			// Zyklisch auf neue Daten pollen
			fbReceiveDataBytes(
				pPrefix				:= ADR(stOptionsIntern.sPrefix),
				LenPrefix			:= stOptionsIntern.nLenPrefix,
				pSuffix				:= ADR(stOptionsIntern.sSuffix),
				LenSuffix			:= stOptionsIntern.nLenSuffix,
				
				Timeout				:= stOptionsIntern.tTimeTimeout,
				Reset					:= FALSE ,
				
				pReceiveData		:= ADR(stRxStringBuffer),
				SizeReceiveData	:= SIZEOF(stRxStringBuffer)-1,
				RXbuffer				:= stRxBuffer
			);

			IF fbReceiveDataBytes.Error <> 0
			THEN	// Fehler beim Datenempfangen
				nRxCount					:= 0;
				bNeueDatenEmpfangen	:= TRUE;
				ccl_Receive.bBusy		:= FALSE;
				ccl_Receive.bDone		:= TRUE;
				ccl_Receive.bError	:= TRUE;
				ccl_Receive.nErrorId	:= fbReceiveDataBytes.Error;
			ELSE

				IF fbReceiveDataBytes.DataReceived
				THEN	// Alle Daten wurden erfolgreich empfangen
				
					nRxCount	:= UDINT_TO_INT(fbReceiveDataBytes.LenReceiveData);
					IF nRxCount <= cBufferSize_StringBuffer
					THEN
						stRxStringBuffer.sData:=LEFT(stRxStringBuffer.sData,nRxCount);
					ELSE
						stRxStringBuffer.sData:=LEFT(stRxStringBuffer.sData,cBufferSize_StringBuffer);
					END_IF
					stRxStringBuffer:= nccl_ReceiveBarcode(stRxStringBuffer);
					nRxCount:=LEN(stRxStringBuffer.sData);

					bRxTimeout:= fbReceiveDataBytes.RxTimeout;
					bNeueDatenEmpfangen	:= TRUE;
				END_IF;
			END_IF
	END_CASE

	// Empfang Oberflaeche. Darauf warten, die die Oberfäche das Bit zurück setzt.
	IF	bNeueDatenEmpfangen
		AND stOptions.nCommVB = 1
	THEN
		bWartenAufVBA_HMI	:= TRUE;
	END_IF

END_IF
END_METHOD

METHOD FB_init : BOOL
VAR_INPUT
	bInitRetains	: BOOL; // if TRUE, the retain variables are initialized (warm start / cold start)
	bInCopyCode		: BOOL;  // if TRUE, the instance afterwards gets moved into the copy code (online change)
	
	I_Options		: ST_ComPortOptions;	
END_VAR
stOptions	:= I_Options;
END_METHOD

METHOD PUBLIC nccl_Config : ST_MethodResult	// Methode muss so lange aufgerufen werden, bis True zurück gibt
// Konfigruation der Klemmen

CASE stOptions.ePort OF
	// PC-ComPort kann man nicht aus der PLC heraus konfigurieren
	E_ComPortHardware.cComportPc:
	
		nccl_Config.bDone	:= TRUE;

	// EL-Klemmen Konfigurieren
	E_ComPortHardware.cComportEL:
	
		CASE nConfigState OF
			
			0:  // Baudrate schreiben, dafür wird mit nWordBuffer die Zeile der Dropdownliste errechnet, die dann geschrieben wird. Es wird nicht direkt die Baudrate geschrieben.(Wäre ja auch zu einfach)
				nccl_Config.bBusy	:= TRUE;
				nIndex:=16#4073;
				nSubIndex:=0;

				nWordBuffer	:= 4;
				nTmpVar		:= stOptions.nBaudrate;
				
				// Ist die Baudrate bei min(1200) angelangt, ist fertig berechnet
				WHILE nTmpVar > 2400 DO
					nTmpVar		:= nTmpVar/2;
					nWordBuffer	:= nWordBuffer+1;
				END_WHILE

				fbEcCoWrite(
					sNetId		:= F_CreateAmsNetId(stComPortIn.stInfoData.stADSNetId) ,
					nSlaveAddr	:= stComPortIn.stInfoData.nADSPort,

					nSubIndex	:= nSubIndex,
					nIndex		:= nIndex,

					pSrcBuf		:= ADR(nWordBuffer),
					cbBufLen		:= SIZEOF(nWordBuffer),
					bExecute		:= NOT fbEcCoWrite.bBusy,
					tTimeout		:= T#3S
				);

			1:  // Frame
				nccl_Config.bBusy	:= TRUE;
				nIndex:=16#4074;
				nSubIndex:=0;

				IF stOptions.nDatenbits = 7
				THEN
					IF stOptions.nStopbits = 1
					THEN
						(*7x1 *)
						CASE stOptions.nParitaet OF
							PARITY_NONE	: nWordBuffer	:= 1;
							PARITY_EVEN	: nWordBuffer	:= 1;
							PARITY_ODD	: nWordBuffer	:= 2;
						END_CASE
					ELSE
						(*7x2 *)
						CASE stOptions.nParitaet OF
							PARITY_NONE	: nWordBuffer	:= 9;
							PARITY_EVEN	: nWordBuffer	:= 9;
							PARITY_ODD	: nWordBuffer	:= 10;
						END_CASE
					END_IF
				ELSE
					(*8x1 *)
					IF stOptions.nStopbits = 1 THEN
						CASE stOptions.nParitaet OF
							PARITY_NONE	: nWordBuffer	:= 3;
							PARITY_EVEN	: nWordBuffer	:= 4;
							PARITY_ODD	: nWordBuffer	:= 5;
						END_CASE
					ELSE
						(*8x2 *)
						CASE stOptions.nParitaet OF
							PARITY_NONE	: nWordBuffer	:= 11;
							PARITY_EVEN	: nWordBuffer	:= 12;
							PARITY_ODD	: nWordBuffer	:= 13;
						END_CASE
					END_IF
				END_IF

				fbEcCoWrite(
					sNetId		:= F_CreateAmsNetId(stComPortIn.stInfoData.stADSNetId) ,
					nSlaveAddr	:= stComPortIn.stInfoData.nADSPort,

					nSubIndex	:= nSubIndex,
					nIndex		:= nIndex,

					pSrcBuf		:= ADR(nWordBuffer),
					cbBufLen		:= SIZEOF(nWordBuffer),
					bExecute		:= NOT fbEcCoWrite.bBusy,
					tTimeout		:= T#3S
				);

			2:  // Handshake RTS/CTS
				nccl_Config.bBusy	:= TRUE;
				nIndex		:= 16#4075;
				nSubIndex	:= 1;

				IF stOptions.nHandshake = HANDSHAKE_RTSCTS
				THEN
					bBuffer:=TRUE;
				ELSE
					bBuffer:=FALSE;
				END_IF

				fbEcCoWrite(
					sNetId		:= F_CreateAmsNetId(stComPortIn.stInfoData.stADSNetId) ,
					nSlaveAddr	:= stComPortIn.stInfoData.nADSPort,

					nSubIndex	:= nSubIndex,
					nIndex		:= nIndex,

					pSrcBuf		:= ADR(bBuffer),
					cbBufLen		:= SIZEOF(bBuffer),
					bExecute		:= NOT fbEcCoWrite.bBusy,
					tTimeout		:= T#3S
				);

			3:  (* XON/XOFF tx *)
				nccl_Config.bBusy	:= TRUE;
				nIndex		:= 16#4075;
				nSubIndex	:= 2;

				IF stOptions.nHandshake = HANDSHAKE_XONXOFF
				THEN
					bBuffer:=TRUE;
				ELSE
					bBuffer:=FALSE;
				END_IF

				fbEcCoWrite(
					sNetId		:= F_CreateAmsNetId(stComPortIn.stInfoData.stADSNetId) ,
					nSlaveAddr	:= stComPortIn.stInfoData.nADSPort,

					nSubIndex	:= nSubIndex,
					nIndex		:= nIndex,

					pSrcBuf		:= ADR(bBuffer),
					cbBufLen		:= SIZEOF(bBuffer),
					bExecute		:= NOT fbEcCoWrite.bBusy,
					tTimeout		:= T#3S
				);

			4:  (* XON/XOFF rx *)
				nccl_Config.bBusy	:= TRUE;
				nIndex		:= 16#4075;
				nSubIndex	:= 3;

				IF stOptions.nHandshake = HANDSHAKE_XONXOFF
				THEN
					bBuffer	:= TRUE;
				ELSE
					bBuffer	:= FALSE;
				END_IF

				fbEcCoWrite(
					sNetId		:= F_CreateAmsNetId(stComPortIn.stInfoData.stADSNetId) ,
					nSlaveAddr	:= stComPortIn.stInfoData.nADSPort,

					nSubIndex	:= nSubIndex,
					nIndex		:= nIndex,

					pSrcBuf		:= ADR(bBuffer),
					cbBufLen		:= SIZEOF(bBuffer),
					bExecute		:= NOT fbEcCoWrite.bBusy,
					tTimeout		:= T#3S
				);
				
		END_CASE

		IF NOT fbEcCoWrite.bBusy
		THEN
			// Bei Fehler ErrorId speichern und Config abbrechen
			IF fbEcCoWrite.bError
			THEN
				nccl_Config.nErrorId	:= UDINT_TO_INT(fbEcCoWrite.nErrId);
			ELSE
				IF nConfigState < 4
				THEN
					nConfigState	:= nConfigState+1;
				ELSE
					nccl_Config.bBusy	:= FALSE;
					nccl_Config.bDone	:= TRUE;	// Konfiguration ist fertig!!!
				END_IF
			END_IF

		END_IF
		
		nccl_Config.bError	:= fbEcCoWrite.bError;
		nccl_Config.nErrorId	:= UDINT_TO_INT(fbEcCoWrite.nErrId);

	// KL-Klemmen Konfigurieren
	E_ComPortHardware.cComportKL:
	
		CASE stOptions.eComPortBytes OF
			
			E_ComPortKlemmenBytes.cComport3Bytes:
			
				fbComPortKL6configuration(
					Execute		:= NOT fbComPortKL6configuration.Busy,
					Mode			:= SERIALLINEMODE_KL6_3B_ALTERNATIVE,
					Baudrate		:= stOptions.nBaudrate,
					NoDatabits	:= UDINT_TO_BYTE(stOptions.nDatenbits),
					Parity		:= stOptions.nParitaet,
					Stopbits		:= UDINT_TO_BYTE(stOptions.nStopbits),
					Handshake	:= stOptions.nHandshake,
					pCOMin		:= ADR(stComPortIn.stKlemmeIn3B),
					pCOMout		:= ADR(stComPortOut.stKlemmeOut3B),
					SizeComIn	:= SIZEOF(stComPortIn.stKlemmeIn3B)
				);
				
				nccl_Config.bBusy		:= fbComPortKL6configuration.Busy;
				nccl_Config.bDone		:= fbComPortKL6configuration.Done;
				nccl_Config.bError	:= fbComPortKL6configuration.Error;
				nccl_Config.nErrorId	:= fbComPortKL6configuration.ErrorId;

			E_ComPortKlemmenBytes.cComport5Bytes:
			
				fbComPortKL6configuration(
					Execute		:= NOT fbComPortKL6configuration.Busy ,
					Mode			:= SERIALLINEMODE_KL6_5B_STANDARD,
					Baudrate		:= UINT_TO_UDINT(stOptions.nBaudrate),
					NoDatabits	:= UDINT_TO_BYTE(stOptions.nDatenbits),
					Parity		:= stOptions.nParitaet,
					Stopbits		:= UDINT_TO_BYTE(stOptions.nStopbits),
					Handshake	:= stOptions.nHandshake,
					pCOMin		:= ADR(stComPortIn.stKlemmeIn5B),
					pCOMout		:= ADR(stComPortOut.stKlemmeOut5B),
					SizeComIn	:= SIZEOF(stComPortIn.stKlemmeIn5B)
				);
				
				nccl_Config.bBusy		:= fbComPortKL6configuration.Busy;
				nccl_Config.bDone		:= fbComPortKL6configuration.Done;
				nccl_Config.bError	:= fbComPortKL6configuration.Error;
				nccl_Config.nErrorId	:= fbComPortKL6configuration.ErrorId;

			E_ComPortKlemmenBytes.cComport22Bytes:
			
				fbComPortKL6configuration(
					Execute		:= NOT fbComPortKL6configuration.Busy ,
					Mode 			:= SERIALLINEMODE_KL6_22B_STANDARD,
					Baudrate		:= UDINT_TO_UINT(stOptions.nBaudrate),
					NoDatabits	:= UDINT_TO_BYTE(stOptions.nDatenbits),
					Parity		:= stOptions.nParitaet,
					Stopbits		:= UDINT_TO_BYTE(stOptions.nStopbits),
					Handshake	:= stOptions.nHandshake,
					pCOMin		:= ADR(stComPortIn.stKlemmeIn22B),
					pCOMout		:= ADR(stComPortOut.stKlemmeOut22B),
					SizeComIn	:= SIZEOF(stComPortIn.stKlemmeIn22B)
				);
				
				nccl_Config.bBusy		:= fbComPortKL6configuration.Busy;
				nccl_Config.bDone		:= fbComPortKL6configuration.Done;
				nccl_Config.bError	:= fbComPortKL6configuration.Error;
				nccl_Config.nErrorId	:= fbComPortKL6configuration.ErrorId;

		END_CASE
END_CASE;

// Konfiguration in die internen Konfiguration übernehmen
stOptionsIntern.tTimeTimeout	:= UDINT_TO_TIME(stOptions.nTimeout);

// Präfix-Konfiguration
stOptionsIntern.nLenPrefix	:= 0;
stOptionsIntern.sPrefix		:= '';

stOptionsIntern.nPrefix		:= UDINT_TO_BYTE(stOptions.nPrefix);

IF stOptionsIntern.nPrefix > 0
THEN
	stOptionsIntern.nLenPrefix	:= stOptionsIntern.nLenPrefix+1;
	stOptionsIntern.sPrefix		:= CONCAT(stOptionsIntern.sPrefix,CHR(stOptionsIntern.nPrefix));
END_IF

// Suffix-Konfiguration
stOptionsIntern.nLenSuffix	:= 0;
stOptionsIntern.sSuffix		:= '';

stOptionsIntern.arrSuffix[1]	:= UDINT_TO_BYTE(stOptions.nSuffix1);
IF stOptionsIntern.arrSuffix[1] > 0
THEN
	stOptionsIntern.nLenSuffix	:= stOptionsIntern.nLenSuffix+1;
	stOptionsIntern.sSuffix		:= CONCAT(stOptionsIntern.sSuffix,CHR(stOptionsIntern.arrSuffix[1]));
END_IF

stOptionsIntern.arrSuffix[2]	:= UDINT_TO_BYTE(stOptions.nSuffix2);
IF stOptionsIntern.arrSuffix[2] > 0
THEN
	stOptionsIntern.nLenSuffix	:= stOptionsIntern.nLenSuffix+1;
	stOptionsIntern.sSuffix		:= CONCAT(stOptionsIntern.sSuffix,CHR(stOptionsIntern.arrSuffix[2]));

	IF stOptionsIntern.arrSuffix[1] = 0
	THEN
		stOptionsIntern.arrSuffix[1]:= stOptionsIntern.arrSuffix[2];
		stOptionsIntern.arrSuffix[2]:= 0;
	END_IF
END_IF

// Bufferlänge auf bei Überschreiten der max Größe, auf die max Größe setzen
IF stOptions.nLength > cBufferSize_IntBuffer
	OR stOptions.nLength = 0
THEN
	stOptionsIntern.nLength:=cBufferSize_IntBuffer;
ELSE
	stOptionsIntern.nLength:=stOptions.nLength;
END_IF
END_METHOD

METHOD INTERNAL nccl_PrepareSendBarcode : ST_ComPortStringBuffer
VAR_INPUT
	I_stSendString	:	ST_ComPortStringBuffer;
END_VAR
IF stOptionsIntern.nLenPrefix > 0
THEN
	nccl_PrepareSendBarcode.sData:=CONCAT(stOptionsIntern.sPrefix,I_stSendString.sData);
ELSE
	nccl_PrepareSendBarcode	:= I_stSendString;
END_IF

IF stOptionsIntern.nLenSuffix > 0
THEN
	nccl_PrepareSendBarcode.sData:=CONCAT(nccl_PrepareSendBarcode.sData,stOptionsIntern.sSuffix);
END_IF
END_METHOD

METHOD INTERNAL nccl_ReceiveBarcode : ST_ComPortStringBuffer
VAR_INPUT
	I_stReceiveString	: ST_ComPortStringBuffer;
END_VAR

VAR
	nStartPosition	: INT;
	nEndPosition	: INT;
	bPrefixFound	: BOOL;
END_VAR
nStartPosition	:= 0;
IF stOptionsIntern.nLenPrefix = 0
THEN
	bPrefixFound:=TRUE;
ELSE
	bPrefixFound:=FALSE;

	REPEAT
		nStartPosition	:= FIND(I_stReceiveString.sData,stOptionsIntern.sPrefix);
		IF nStartPosition > 0
		THEN
			bPrefixFound:=TRUE; (* Mindesten 1 x Prefix *)

			nStartPosition	:= nStartPosition + stOptionsIntern.nLenPrefix;
			I_stReceiveString.sData	:= MID(I_stReceiveString.sData,LEN(I_stReceiveString.sData)-nStartPosition+1,nStartPosition);
		END_IF
	UNTIL
		nStartPosition = 0
	END_REPEAT
END_IF

IF bPrefixFound
THEN
	nEndPosition:=0;

	IF stOptionsIntern.nLenSuffix = 0
	THEN
		nEndPosition	:= LEN(I_stReceiveString.sData);
	ELSE
		nEndPosition	:= FIND(I_stReceiveString.sData,stOptionsIntern.sSuffix)-1;
	END_IF

	IF nEndPosition > 0
	THEN
		nccl_ReceiveBarcode.sData	:= MID(I_stReceiveString.sData,nEndPosition,1);
	END_IF
END_IF
END_METHOD

METHOD PUBLIC nccl_Reset : BOOL
VAR
	nRxBufferIndx	: INT;
	fbClearBuffer	: ClearComBuffer;
END_VAR
// Reset
IF NOT stConfigResult.bBusy
THEN
	bNeueDatenEmpfangen	:= FALSE;
	bWartenAufVBA_HMI		:= FALSE;
	bRxTimeout				:=FALSE;

	// Empfangsdaten löschen
	FOR nRxBufferIndx	:= 0 TO cBufferSize_IntBuffer
	DO
		stRxIntBuffer.arrData[nRxBufferIndx]:=0;
	END_FOR

	stRxStringBuffer.sData:='';
	
	// internen Empfangspuffer löschen
	fbClearBuffer(Buffer:=stRxBuffer);

	// Empfangsbaustein für Datenstream resetten
	fbReceiveDataBytes(
		Reset				:= TRUE ,
		pReceiveData	:= ADR(stRxByteBuffer),
		RXbuffer			:= stRxBuffer
	);

	// interne Empfangs- und Sendepuffer nochmals händisch löschen- 
	stTxBuffer.Count:=0;
	stTxBuffer.RdIdx:=0;
	stTxBuffer.WrIdx:=0;
	stTxBuffer.Error:=0;

	stRxBuffer.Count:=0;
	stRxBuffer.RdIdx:=0;
	stRxBuffer.WrIdx:=0;
	stRxBuffer.Error:=0;

	// Diagnose zurücksetzen
	nDiagRxCycleCounter	:=0;
	nDiagRxErrorCounter	:=0;
	nDiagRxLastErrorId	:=0;
	nDiagRxDataCounter	:=0;

	sTmpDiagMessage	:= CONCAT('RxCycle:', UINT_TO_STRING(nDiagRxCycleCounter));
	sTmpDiagMessage	:= CONCAT(sTmpDiagMessage, CONCAT(' - RxData:', INT_TO_STRING(nDiagRxDataCounter)));
	sTmpDiagMessage	:= CONCAT(sTmpDiagMessage, CONCAT(' - RxError:', UINT_TO_STRING(nDiagRxErrorCounter)));
	sTmpDiagMessage	:= CONCAT(sTmpDiagMessage, CONCAT(' - RxErrorId:', INT_TO_STRING(nDiagRxLastErrorId)));
	sDiagMessage		:= sTmpDiagMessage;

	bStartPLC	:= FALSE;	// Config auslösen
	nccl_Reset	:= TRUE;	// Resetten fertig
END_IF
END_METHOD

{attribute 'hide_all_locals'}
METHOD PUBLIC nccl_Send : ST_MethodResult	// Methode ist innerhalb eines Zyklusses fertig.
VAR_INPUT
	I_stTxIntBuffer			: ST_ComPortIntBuffer;	// Int Uebergabepuffer
	I_stTxStringBuffer		: ST_ComPortStringBuffer;	// String Uebergabepuffer

	I_nTxCount					: INT;	// Anzahl zu sendender Zeichen
	I_eTxProtokoll				: E_ComPortProtokoll	:= E_ComPortProtokoll.cProtokollNone;	// Sendenprotokoll
END_VAR
VAR
	nTxBufferIndx				: INT;
	stBarcodeTxStringBuffer	: ST_ComPortStringBuffer;
	
	eProtokoll					: E_ComPortProtokoll;
	stTxByteBuffer				: Tc2_SerialCom.P3964buffer;
	fbSendByteDirect			: Tc2_SerialCom.SendByte;
	fbSendDataBytes			: Tc2_SerialCom.SendData;
END_VAR
// Senden
IF stOptions.nAktiv = 1
	AND NOT stConfigResult.bBusy
THEN
	nccl_Send.bBusy	:= TRUE;	// pauschal auf busy setzen

	IF I_eTxProtokoll <> E_ComPortProtokoll.cProtokollNone
	THEN
		eProtokoll := I_eTxProtokoll;
	ELSE
		eProtokoll := stOptions.eProtokoll;
	END_IF

	CASE eProtokoll OF
		E_ComPortProtokoll.cProtokollNone:
			;	// Ohne Protokoll nix machen
			
		E_ComPortProtokoll.cProtokollData:
			
			nTxBufferIndx:=0;
			WHILE nTxBufferIndx < I_nTxCount
				AND nTxBufferIndx <= cBufferSize_IntBuffer
			DO
				stTxByteBuffer.D[nTxBufferIndx]	:= UINT_TO_BYTE(I_stTxIntBuffer.arrData[nTxBufferIndx]);
				nTxBufferIndx	:= nTxBufferIndx+1;
			END_WHILE

			fbSendDataBytes(
				pSendData:= ADR(stTxByteBuffer),
				Length	:= INT_TO_UDINT(I_nTxCount),
				TXbuffer	:= stTxBuffer);

			// Sendefehler
			IF  fbSendDataBytes.Error <> 0
			THEN
				nccl_Send.nErrorId	:= fbSendDataBytes.Error;
				nccl_Send.bError	:= TRUE; 
				nccl_Send.bBusy	:= FALSE;
			ELSE	// Erfolgreich gesendet
				IF NOT fbSendDataBytes.Busy
				THEN
					nccl_Send.bBusy	:= FALSE;
					nccl_Send.bDone	:= TRUE;
				END_IF
			END_IF

		E_ComPortProtokoll.cProtokollDirect:
			
			nTxBufferIndx := 0;
			IF I_nTxCount > cBufferSize_IntBuffer
			THEN
				I_nTxCount := cBufferSize_IntBuffer;
			END_IF

			WHILE nTxBufferIndx < I_nTxCount
				AND fbSendByteDirect.Error = 0
			DO
				fbSendByteDirect(
					SendByte	:= UINT_TO_BYTE(I_stTxIntBuffer.arrData[nTxBufferIndx]),
					TXbuffer	:= stTxBuffer
				);
				nTxBufferIndx	:= nTxBufferIndx+1;
				
			END_WHILE

			// Sendefehler
			IF  fbSendByteDirect.Error <> 0
			THEN
				nccl_Send.nErrorId	:= fbSendByteDirect.Error;
				nccl_Send.bError	:= TRUE; 
				nccl_Send.bBusy	:= FALSE;
			ELSE	// Erfolgreich gesendet
				IF NOT fbSendByteDirect.Busy
				THEN
					nccl_Send.bBusy	:= FALSE;
					nccl_Send.bDone	:= TRUE;
				END_IF
			END_IF

		E_ComPortProtokoll.cProtokollBarcode:
			
			stBarcodeTxStringBuffer	:= nccl_PrepareSendBarcode(I_stTxStringBuffer);

			fbSendDataBytes(
				pSendData	:= ADR(stBarcodeTxStringBuffer),
				Length		:= INT_TO_BYTE(LEN(stBarcodeTxStringBuffer.sData)),
				TXbuffer		:= stTxBuffer);

			// Sendefehler
			IF  fbSendDataBytes.Error <> 0
			THEN
				nccl_Send.nErrorId	:= fbSendDataBytes.Error;
				nccl_Send.bError		:= TRUE; 
				nccl_Send.bBusy		:= FALSE;
			ELSE	// Erfolgreich gesendet
				IF NOT fbSendDataBytes.Busy
				THEN
					nccl_Send.bBusy	:= FALSE;
					nccl_Send.bDone	:= TRUE;
				END_IF
			END_IF
	END_CASE
END_IF

stSendResult	:= nccl_Send;
END_METHOD

PROPERTY PUBLIC P_bDatenVorhanden : BOOL
GET
P_bDatenVorhanden	:= bNeueDatenEmpfangen;
END_GET
END_PROPERTY

// Liest die Empfangenen Daten aus und setzt das Empfangsbit zurück
PROPERTY PUBLIC P_stEmpfangeneDaten : ST_ComPortIntBuffer
GET
P_stEmpfangeneDaten	:= stRxIntBuffer;
bNeueDatenEmpfangen	:= FALSE;
END_GET
END_PROPERTY

// Liest die Empfangenen Daten aus und setzt das Empfangsbit zurück
PROPERTY PUBLIC P_stEmpfangenerString : STRING
GET
P_stEmpfangenerString	:= stRxStringBuffer.sData;
bNeueDatenEmpfangen		:= FALSE;
END_GET
END_PROPERTY

END_FUNCTION_BLOCK

// POUs/DiagSafety/FB_DiagEL2904
// OBSOLET, wenn man FB_TwinSAFEKlemmenInfo benutzt
FUNCTION_BLOCK FB_DiagEL2904
VAR_INPUT
	I_stEcAdsAddr			: AMSADDR;
	I_nDiag					: USINT;
	I_strBMK					: STRING;
END_VAR
VAR_OUTPUT
	Q_stTemperatur 		: ST_EL2904Temp;
	Q_bError					: BOOL;
	Q_strDiag				: STRING;
END_VAR
VAR
	nStep					: INT;
	nLastStep			: INT;
	tonReadDiag			: TON;
	fbEcCoeSdoRead		: FB_EcCoESdoReadEx;
	stDiagObject		: ST_EL2904Diag;
	nDiag0_3				: BYTE;
	strDiag				: STRING;
END_VAR


act_Diag();
act_DiagObjekte();

IF strDiag <> ''
THEN
	Q_strDiag 	:= CONCAT(I_strBMK,CONCAT(' ',strDiag));
	Q_bError		:= TRUE;
ELSE
	Q_bError		:= FALSE;
END_IF

ACTION act_Diag:

strDiag:='';

IF I_nDiag.4 
THEN
	strDiag	:= 'Fehler beim FSoE Slave erkannt | '; 
END_IF

IF I_nDiag.5 
THEN
	strDiag	:= CONCAT(strDiag,'FSoE Slave meldet Failsafe Value aktiv | ');
END_IF

IF I_nDiag.6 
THEN
	strDiag	:= CONCAT(strDiag,'StartUp | ');
END_IF

IF I_nDiag.7 
THEN
	strDiag	:= CONCAT(strDiag, 'FSoE Master meldet Failsafe Value aktiv | ');
END_IF
	
nDiag0_3 := USINT_TO_BYTE(I_nDiag) AND 16#0F;

CASE nDiag0_3 OF
	1:		strDiag	:= CONCAT(strDiag,'Ungültiges Kommando | ');
	2:		strDiag	:= CONCAT(strDiag,'Unbekanntes Kommando | ');
	3:		strDiag	:= CONCAT(strDiag,'Ungültige Connection ID | ');
	4:		strDiag	:= CONCAT(strDiag,'Ungültige CRC | ');
	5:		strDiag	:= CONCAT(strDiag,'Watchdog abgelaufen | ');
	6:		strDiag	:= CONCAT(strDiag,'Ungültige FSoE Adresse | ');
	7:		strDiag	:= CONCAT(strDiag,'Ungültige Daten | ');
	8:		strDiag	:= CONCAT(strDiag,'Ungültige Kommunikationsparameterlänge | ');
	9:		strDiag	:= CONCAT(strDiag,'Ungültige Kommunikationsparameter | ');
	10:	strDiag	:= CONCAT(strDiag,'Ungültige Anwenderparameterlänge | ');
	11:	strDiag	:= CONCAT(strDiag,'Ungültige Anwenderparameter | ');
	12:	strDiag	:= CONCAT(strDiag,'FSoE Master Reset | ');
	13:	strDiag	:= CONCAT(strDiag,'Modulfehler auf Slave erkannt, bei aktivierter Option "Modulfehler ist ComError" | ');
	14:	strDiag	:= CONCAT(strDiag,'Modulfehler auf EL290x erkannt, bei aktivierter Option "Error acknowledge active" | ');
	15:	strDiag	:= CONCAT(strDiag,'Slave noch nicht gestartet, oder unerwartetes Fehlerargument | ');
END_CASE

IF stDiagObject.nErrorOutputs.0
THEN
	strDiag	:= CONCAT(strDiag,'Fremdeinspeisung oder Querschluss am Ausgang 1');
ELSIF  stDiagObject.nErrorOutputs.1 
THEN
	strDiag	:= CONCAT(strDiag,'Fremdeinspeisung oder Querschluss am Ausgang 2');
ELSIF  stDiagObject.nErrorOutputs.2
THEN
	strDiag	:= CONCAT(strDiag,'Fremdeinspeisung oder Querschluss am Ausgang 3');
ELSIF  stDiagObject.nErrorOutputs.3 
THEN
	strDiag	:= CONCAT(strDiag,'Fremdeinspeisung oder Querschluss am Ausgang 4');
ELSIF  stDiagObject.nErrorOutputs.4 
THEN
	strDiag	:= CONCAT(strDiag,'Ausgangsstrom < 20mA oder > 500mA am Ausgang 1');
ELSIF  stDiagObject.nErrorOutputs.5
THEN
	strDiag	:= CONCAT(strDiag,'Ausgangsstrom < 20mA oder > 500mA am Ausgang 2');
ELSIF  stDiagObject.nErrorOutputs.6 
THEN
	strDiag	:= CONCAT(strDiag,'Ausgangsstrom < 20mA oder > 500mA am Ausgang 3');
ELSIF  stDiagObject.nErrorOutputs.7 
THEN
	strDiag	:= CONCAT(strDiag,'Ausgangsstrom < 20mA oder > 500mA am Ausgang 4');
	
ELSIF stDiagObject.nSupplyError.0
THEN
	strDiag	:= CONCAT(strDiag,'Feldspannung zu hoch');
ELSIF stDiagObject.nSupplyError.1
THEN
	strDiag	:= CONCAT(strDiag,'Feldspannung zu niedrig');
	
ELSIF stDiagObject.nTemperatureError.0
THEN
	strDiag	:= CONCAT(strDiag,'Übertemperatur µC1');
ELSIF stDiagObject.nTemperatureError.1
THEN
	strDiag	:= CONCAT(strDiag,'Übertemperatur µC2');
ELSIF stDiagObject.nTemperatureError.2
THEN
	strDiag	:= CONCAT(strDiag,'Übertemperatur der Ausgangsplatine');
ELSIF stDiagObject.nTemperatureError.3
THEN
	strDiag	:= CONCAT(strDiag,'Untertemperatur µC1');
ELSIF stDiagObject.nTemperatureError.4
THEN
	strDiag	:= CONCAT(strDiag,'Untertemperatur µC2');
ELSIF stDiagObject.nTemperatureError.5
THEN
	strDiag	:= CONCAT(strDiag,'Untertemperatur der Ausgangsplatine');
ELSIF stDiagObject.nTemperatureError.6
THEN
	strDiag	:= CONCAT(strDiag,'Temperaturdifferenz auf der Prozessorplatine zu groß');
ELSIF stDiagObject.nTemperatureError.7
THEN
	strDiag	:= CONCAT(strDiag,'Temperaturdifferenz zwischen den Platinen zu groß');
END_IF
END_ACTION

ACTION act_DiagObjekte:
CASE nStep OF

0: tonReadDiag(IN:= TRUE,	
					PT :=T#2S);
		fbEcCoeSdoRead(
		bExecute			:= FALSE);
	IF tonReadDiag.Q
	THEN
		nStep := 10;
	END_IF

10:	
	fbEcCoeSdoRead(
		sNetId			:= F_CreateAmsNetId(I_stEcAdsAddr.netId), 
		nSlaveAddr		:= I_stEcAdsAddr.port, 
		nSubIndex		:= 1, 
		nIndex			:= 16#FA80, 
		pDstBuf			:= ADR(Q_stTemperatur), 
		cbBufLen			:= SIZEOF(Q_stTemperatur), 
		bExecute			:= TRUE, 
		tTimeout			:= T#5S, 
		bCompleteAccess:= TRUE );
	
	IF NOT fbEcCoeSdoRead.bBusy
		AND NOT fbEcCoeSdoRead.bError
	THEN
		fbEcCoeSdoRead(bExecute := FALSE);
		nStep := 20;
	ELSIF fbEcCoeSdoRead.bError
	THEN
		nStep := 0;
	END_IF

20: fbEcCoeSdoRead(
		sNetId			:= F_CreateAmsNetId(I_stEcAdsAddr.netId), 
		nSlaveAddr		:= I_stEcAdsAddr.port, 
		nSubIndex		:= 1, 
		nIndex			:= 16#800E, 
		pDstBuf			:= ADR(stDiagObject), 
		cbBufLen			:= SIZEOF(stDiagObject), 
		bExecute			:= TRUE, 
		tTimeout			:= T#5S, 
		bCompleteAccess:= TRUE);
	IF NOT fbEcCoeSdoRead.bBusy
		AND NOT fbEcCoeSdoRead.bError
	THEN
		nStep	:= 0;
	ELSIF fbEcCoeSdoRead.bError
	THEN
		nStep := 0;
	END_IF
END_CASE


IF nStep <> nLastStep
THEN
	tonReadDiag(IN:= FALSE);
	nLastStep := nStep;
END_IF
END_ACTION

END_FUNCTION_BLOCK

// POUs/DiagSafety/FB_DiagEL2912
// OBSOLET, wenn man FB_TwinSAFEKlemmenInfo benutzt
FUNCTION_BLOCK FB_DiagEL2912
VAR_INPUT				
	I_stEcAdsAddr			: AMSADDR;
	I_nDiag					: USINT;
	I_strBMK					: STRING;
END_VAR
VAR_OUTPUT
	Q_bError					: BOOL;
	Q_strDiag				: STRING;
END_VAR
VAR
	nDiag0_3				: BYTE;
	strDiag				: STRING;
END_VAR


act_Diag();

IF strDiag <> ''
THEN
	Q_strDiag 	:= CONCAT(I_strBMK,CONCAT(' ',strDiag));
	Q_bError		:= TRUE;
ELSE
	Q_bError		:= FALSE;
END_IF

ACTION act_Diag:

strDiag:='';

IF I_nDiag.4 
THEN
	strDiag	:= 'Fehler beim FSoE Slave erkannt | '; 
END_IF

IF I_nDiag.5 
THEN
	strDiag	:= CONCAT(strDiag,'FSoE Slave meldet Failsafe Value aktiv | ');
END_IF

IF I_nDiag.6 
THEN
	strDiag	:= CONCAT(strDiag,'StartUp | ');
END_IF

IF I_nDiag.7 
THEN
	strDiag	:= CONCAT(strDiag, 'FSoE Master meldet Failsafe Value aktiv | ');
END_IF
	
nDiag0_3 := USINT_TO_BYTE(I_nDiag) AND 16#0F;

CASE nDiag0_3 OF
	1:		strDiag	:= CONCAT(strDiag,'Ungültiges Kommando | ');
	2:		strDiag	:= CONCAT(strDiag,'Unbekanntes Kommando | ');
	3:		strDiag	:= CONCAT(strDiag,'Ungültige Connection ID | ');
	4:		strDiag	:= CONCAT(strDiag,'Ungültige CRC | ');
	5:		strDiag	:= CONCAT(strDiag,'Watchdog abgelaufen | ');
	6:		strDiag	:= CONCAT(strDiag,'Ungültige FSoE Adresse | ');
	7:		strDiag	:= CONCAT(strDiag,'Ungültige Daten | ');
	8:		strDiag	:= CONCAT(strDiag,'Ungültige Kommunikationsparameterlänge | ');
	9:		strDiag	:= CONCAT(strDiag,'Ungültige Kommunikationsparameter | ');
	10:	strDiag	:= CONCAT(strDiag,'Ungültige Anwenderparameterlänge | ');
	11:	strDiag	:= CONCAT(strDiag,'Ungültige Anwenderparameter | ');
	12:	strDiag	:= CONCAT(strDiag,'FSoE Master Reset | ');
	13:	strDiag	:= CONCAT(strDiag,'Modulfehler auf Slave erkannt, bei aktivierter Option "Modulfehler ist ComError" | ');
	14:	strDiag	:= CONCAT(strDiag,'Modulfehler auf EL290x erkannt, bei aktivierter Option "Error acknowledge active" | ');
	15:	strDiag	:= CONCAT(strDiag,'Slave noch nicht gestartet, oder unerwartetes Fehlerargument | ');
END_CASE
END_ACTION

END_FUNCTION_BLOCK

// POUs/DiagSafety/FB_TwinSAFE_Conn_Info
(* Version arrHistory: 
Description: Ethercat-Saftey Diagnose
Date          | Version    | created under        | Author          | Remark 
---------------------------------------------------------------------------------------- 
12/09/2011    | 1.1.0      | V2.11.0 (Build 1551) | T.Löhner        | first release
*)
FUNCTION_BLOCK FB_TwinSAFE_Conn_Info
VAR_INPUT
	I_stInfoData	: ST_TwinSAFE_Conn_Info;
	I_nGrpId			: INT;
	I_nConnId		: INT;
	I_sConnName		: STRING;
END_VAR
VAR_OUTPUT
	Q_bErrorDiag	: BOOL;
	Q_bErrorState	: BOOL;
	Q_sDiag			: Tc2_System.T_MaxString;
	Q_sState			: Tc2_System.T_MaxString;
END_VAR
VAR
	sConn				: STRING;
	nDiag				: INT;
	sState_old		: Tc2_System.T_MaxString;
	sDiag_old		: Tc2_System.T_MaxString;
	tonStateChange	:TON;
	tonDiagChange	:TON;
END_VAR

	(* ========================================================= *)
	actInfo();

	(* ========================================================= *)

ACTION act_Diag:

	IF Q_sDiag<> sDiag_old THEN
		Q_bErrorDiag	:= FALSE;
	ELSE
		Q_bErrorDiag	:= TRUE;
	END_IF

	tonDiagChange(
		IN:= NOT Q_bErrorDiag,
		PT:=t#500ms);

	IF tonDiagChange.Q THEN
		sDiag_old	:= Q_sDiag;
	END_IF

	Q_sDiag			:= CONCAT('Diagnose: ',Q_sDiag);
	Q_sDiag			:= CONCAT(sConn,Q_sDiag);

	(*BE*)
END_ACTION

ACTION act_State:

	IF Q_sState<> sState_old THEN
		Q_bErrorState	:= FALSE;
	ELSE
		Q_bErrorState	:= TRUE;
	END_IF

	tonStateChange(
		IN:= NOT Q_bErrorState,
		PT:=t#500ms);

	IF tonStateChange.Q THEN
		sstate_old	:= Q_sState;
	END_IF

	Q_sState		:= CONCAT('Status: ',Q_sState);
	Q_sState		:= CONCAT(sConn,Q_sState);

	(*BE*)
END_ACTION

ACTION actInfo:
	(* TwinSAFE-Connection *)
	(* ========================================================= *)
	Q_bErrorState		:= FALSE;
	Q_bErrorDiag		:= FALSE;
	Q_sState			:= '';
	Q_sDiag				:= '';

	sConn				:= CONCAT('TwinSAFE Gruppe',INT_TO_STRING(I_nGrpId));
	sConn				:= CONCAT(sConn,' => ');
	sConn				:= CONCAT(sConn,'Connection');
	sConn				:= CONCAT(sConn,INT_TO_STRING(I_nConnId));
	sConn				:= CONCAT(sConn,' ');
	sConn				:= CONCAT(sConn,I_sConnName);
	sConn				:= CONCAT(sConn,' => ');

	(* ========================================================= *)
	(* State *)
	CASE I_stInfoData.nMapState OF
		100: 	Q_sState 			:='Reset';

		101: 	Q_sState 			:='Session';

		102: 	Q_sState 			:='Connection';

		103: 	Q_sState 			:='Parameter';

		104: 	Q_sState 			:='Data';

		105: 	Q_sState 			:='Shutdown';

	ELSE		Q_sState 			:='undefiniert';
				act_State();
	END_CASE

	(* ========================================================= *)
	(* Diagnose *)
	CASE I_stInfoData.nMapDiag OF
			0: ;
	ELSE
		nDiag	:= WORD_TO_INT(UINT_TO_WORD(I_stInfoData.nMapDiag) AND 16#000F);
		CASE nDiag OF
			1: Q_sDiag			 	:='Ungueltiges Kommando';
				act_Diag();

			2: Q_sDiag 			:='Unbekanntes Kommando';
				act_Diag();

			3: Q_sDiag 			:='Ungueltige Connection ID';
				act_Diag();

			4: Q_sDiag 			:='Ungueltige CRC';
				act_Diag();

			5: Q_sDiag 			:='Watchdog abgelaufen';
				act_Diag();

			6: Q_sDiag 			:='Ungueltige FSoE address';
				act_Diag();

			7: Q_sDiag 			:='Ungueltige data';
				act_Diag();

			8: Q_sDiag 			:='Ungueltige Kommunikationsparameterlaenge';
				act_Diag();

			9: Q_sDiag 			:='Ungueltige Kommunikationsparameter';
				act_Diag();

			10:Q_sDiag 			:='Ungueltige Anwenderparameterlaenge';
				act_Diag();

			11:Q_sDiag 			:='Ungueltige Anwenderparameter';
				act_Diag();

			12:Q_sDiag		 		:='FSoE Master Reset';
				act_Diag();
		END_CASE

		nDiag:=WORD_TO_INT(UINT_TO_WORD(I_stInfoData.nMapDiag) AND 16#00F0);
		nDiag:=SHL(nDiag,4);
		CASE nDiag OF
			1 :Q_sDiag 			:='Fehler beim FSoE erkannt';
				act_Diag();

			2 :Q_sDiag 			:='FSoE Slave meldet Failsafe Value aktiv';
				act_Diag();

			4 :Q_sDiag 			:='StartUp';
				act_Diag();

			8 :Q_sDiag 			:='FSoE Master meldet Failsafe Value akriv';
				act_Diag();
		END_CASE
	END_CASE

	(* ========================================================= *)
END_ACTION

END_FUNCTION_BLOCK

// POUs/DiagSafety/FB_TwinSAFE_FBs_Info
(* Version arrHistory:
Description: Ethercat-Saftey Diagnose
Date          | Version    | created under        | Author          | Remark 
---------------------------------------------------------------------------------------- 
12/09/2011    | 1.1.0      | V2.11.0 (Build 1551) | T.Löhner        | first release
*)
FUNCTION_BLOCK FB_TwinSAFE_FBs_Info
VAR_INPUT
	I_stInfoData				: ST_TwinSAFE_FB_Info;
	I_nGrpId						: INT;		(* Id der TwinSAFE-Gruppe*)
	I_nFBId						: INT;		(* Id des Funktionsbausteins*)
	I_sFBName					: STRING;	(* Name des Funktionsbausteins *)
	I_sNameEinGruppe1			: STRING;	(* Bezeichung der beiden Safety-Inputs der 1.FB-Eingangsgruppe 		=> bei EStop/MachineMonitoring/ConnectionShutdown/Muting/TwoHand*)
	I_sNameEinGruppe2			: STRING;	(* Bezeichung der beiden Safety-Inputs der 2.FB-Eingangsgruppe 		=> bei EStop/MachineMonitoring/ConnectionShutdown/Muting/TwoHand*)
	I_sNameEinGruppe3			: STRING;	(* Bezeichung der beiden Safety-Inputs der 3.FB-Eingangsgruppe 		=> bei EStop/MachineMonitoring/ConnectionShutdown/Muting/TwoHand*)
	I_sNameEinGruppe4			: STRING;	(* Bezeichung der beiden Safety-Inputs der 4.FB-Eingangsgruppe 		=> bei EStop/MachineMonitoring/ConnectionShutdown/Muting/TwoHand*)
	I_sNameSecGruppe			: STRING;	(* Bezeichung der beiden Safety-Inputs der FB-Secure-Eingangsgruppe 	=> bei MachineMonitoring *)
	I_sNameEMD1					: STRING;	(* Bezeichung des Safety-Inputs für den Rückführkreis EDM1 				=> bei EStop/MachineMonitoring/Muting *)
	I_sNameEMD2					: STRING;	(* Bezeichung des Safety-Inputs für den Rückführkreis EDM2 				=> bei EStop/MachineMonitoring/Muting *)
	I_sNameOSSDEinGruppe		: STRING;	(* Bezeichung des Safety-Inputs für die OSSD-Eingangsgruppe				=> bei Muting*)
END_VAR

VAR_OUTPUT
	Q_bErrorDiag		: BOOL;					(* Diagnose-Fehler*)
	Q_bErrorState		: BOOL;					(* State-Fehler*)
	Q_sDiag				: Tc2_System.T_MaxString;			(* Diagnose-Fehlerbezeichnung*)
	Q_sState				: Tc2_System.T_MaxString;			(* Diagnose-Fehlerbezeichnung*)
END_VAR

VAR
	sFB				:STRING;
	sState_old		:Tc2_System.T_MaxString;
	sDiag_old		:Tc2_System.T_MaxString;
	tonStateChange	:TON;
	tonDiagChange	:TON;
END_VAR

	(* ========================================================= *)
	;
	(* ========================================================= *)
	(* Aktionsaufrufe erfolgen je nach Art des TwinSAFE-Funktions-
		bausteins beim Aufruf von diesem FB *)

ACTION act_Diag:

	IF Q_sDiag<> sDiag_old THEN
		Q_bErrorDiag	:= FALSE;
	ELSE
		Q_bErrorDiag	:= TRUE;
	END_IF

	tonDiagChange(
		IN:= NOT Q_bErrorDiag,
		PT:=t#500ms);

	IF tonDiagChange.Q THEN
		sDiag_old	:= Q_sDiag;
	END_IF

	Q_sDiag			:= CONCAT('Diagnose: ',Q_sDiag);
	Q_sDiag			:= CONCAT(sFB,Q_sDiag);

	(*BE*)
END_ACTION

ACTION act_State:

	IF Q_sState<> sState_old THEN
		Q_bErrorState	:= FALSE;
	ELSE
		Q_bErrorState	:= TRUE;
	END_IF

	tonStateChange(
		IN:= NOT Q_bErrorState,
		PT:= t#500ms);

	IF tonStateChange.Q THEN
		sstate_old	:= Q_sState;
	END_IF

	Q_sState		:= CONCAT('Status: ',Q_sState);
	Q_sState		:= CONCAT(sFB,Q_sState);

	(*BE*)
END_ACTION

ACTION actInfoAND:
	(* TwinSAFE-Funktionsbaustein FB AND*)
	(* ========================================================= *)
	Q_bErrorState		:= FALSE;
	Q_bErrorDiag		:= FALSE;
	Q_sState			:= '';
	Q_sDiag				:= '';

	sFB				:= CONCAT('TwinSAFE Gruppe',INT_TO_STRING(I_nGrpId));
	sFB				:= CONCAT(sFB,' => ');
	sFB				:= CONCAT(sFB,'FB');
	sFB				:= CONCAT(sFB,INT_TO_STRING(I_nFBId));
	sFB				:= CONCAT(sFB,' ');
	sFB				:= CONCAT(sFB,I_sFBName);
	sFB				:= CONCAT(sFB,' => ');

	(* ========================================================= *)
	(* State *)
	CASE I_stInfoData.nMapState OF
		0:	Q_sState		:= 'undefiniert';
			act_State();

		1:	Q_sState		:= 'Run';

		2:	Q_sState		:= 'Stop';

		3:	Q_sState		:= 'Safe';

	ELSE	Q_sState		:= 'Error';
			act_State();
	END_CASE

	(* ========================================================= *)
	(* Diagnose *)
	(*	stInfoData.uiMapDiag	immer gleich 0*)
	CASE I_stInfoData.nMapState OF
		0:	;
	END_CASE

	(* ========================================================= *)
	(*BE*)
END_ACTION

ACTION actInfoConnectionShutDown:
	(* TwinSAFE-Funktionsbaustein FB Connection Shutdown *)
	(* ========================================================= *)
	Q_bErrorState		:= FALSE;
	Q_bErrorDiag		:= FALSE;
	Q_sState			:= '';
	Q_sDiag				:= '';

	sFB				:= CONCAT('TwinSAFE Gruppe',INT_TO_STRING(I_nGrpId));
	sFB				:= CONCAT(sFB,' => ');
	sFB				:= CONCAT(sFB,'FB');
	sFB				:= CONCAT(sFB,INT_TO_STRING(I_nFBId));
	sFB				:= CONCAT(sFB,' ');
	sFB				:= CONCAT(sFB,I_sFBName);
	sFB				:= CONCAT(sFB,' => ');

	(* ========================================================= *)
	(* State *)
	CASE I_stInfoData.nMapState OF
		0:	Q_sState		:= 'undefiniert';
			act_State();

		2:	Q_sState		:= 'Stop';

		3:	Q_sState		:= 'Safe';

		4:	Q_sState		:= 'Error';
			act_State();

		5:	Q_sState		:= 'Reset';

		10:Q_sState		:= 'Active';

		11:Q_sState		:= 'Deactive';

	ELSE	Q_sState		:= 'Error';
			act_State();
	END_CASE

	(* ========================================================= *)
	(* Diagnose *)
	(*	stInfoData.uiMapDiag	immer gleich 0*)
	CASE I_stInfoData.nMapDiag OF
		0: Q_sDiag :='-';
	ELSE
		IF I_stInfoData.nMapDiag.0 THEN
			Q_sDiag	:='Diskrepanz Fehler Eingangsgruppe 1 => Safety Input => ';
			Q_sDiag	:= CONCAT(Q_sDiag,I_sNameEinGruppe1);
			act_Diag();
		END_IF
	END_CASE

	(* ========================================================= *)
	(*BE*)
END_ACTION

ACTION actInfoDecoupler:
	(* TwinSAFE-Funktionsbaustein FB Decouple*)
	(* ========================================================= *)
	Q_bErrorState		:= FALSE;
	Q_bErrorDiag		:= FALSE;
	Q_sState			:= '';
	Q_sDiag				:= '';

	sFB				:= CONCAT('TwinSAFE Gruppe',INT_TO_STRING(I_nGrpId));
	sFB				:= CONCAT(sFB,' => ');
	sFB				:= CONCAT(sFB,'FB');
	sFB				:= CONCAT(sFB,INT_TO_STRING(I_nFBId));
	sFB				:= CONCAT(sFB,' ');
	sFB				:= CONCAT(sFB,I_sFBName);
	sFB				:= CONCAT(sFB,' => ');

	(* ========================================================= *)
	(* State *)
	CASE I_stInfoData.nMapState OF
		0:	Q_sState		:= 'undefiniert';
			act_State();

		1:	Q_sState		:= 'Run';

		2:	Q_sState		:= 'Stop';

	ELSE	Q_sState		:= 'Error';
			act_State();
	END_CASE

	(* ========================================================= *)
	(* Diagnose *)
	(*	stInfoData.uiMapDiag	immer gleich 0*)
	CASE I_stInfoData.nMapState OF
		0:	;
	END_CASE

	(* ========================================================= *)
	(*BE*)
END_ACTION

ACTION actInfoEDM:
	(* TwinSAFE-Funktionsbaustein FB EDM *)
	(* ========================================================= *)
	Q_bErrorState		:= FALSE;
	Q_bErrorDiag		:= FALSE;
	Q_sState			:= '';
	Q_sDiag				:= '';

	sFB				:= CONCAT('TwinSAFE Gruppe',INT_TO_STRING(I_nGrpId));
	sFB				:= CONCAT(sFB,' => ');
	sFB				:= CONCAT(sFB,'FB');
	sFB				:= CONCAT(sFB,INT_TO_STRING(I_nFBId));
	sFB				:= CONCAT(sFB,' ');
	sFB				:= CONCAT(sFB,I_sFBName);
	sFB				:= CONCAT(sFB,' => ');

	(* ========================================================= *)
	(* State *)
	CASE I_stInfoData.nMapState OF
		0:	Q_sState		:= 'undefiniert';
			act_State();

		2:	Q_sState		:= 'Stop';

		4:	Q_sState		:= 'Error';
			act_State();

		5:	Q_sState		:= 'Reset';

		14:Q_sState		:= 'MON_OFF';

		15:Q_sState		:= 'MON_ON';

	ELSE	Q_sState		:= 'Error';
			act_State();
	END_CASE

	(* ========================================================= *)
	(* Diagnose *)
	CASE I_stInfoData.nMapDiag OF
		0: ;
	ELSE
		IF I_stInfoData.nMapDiag.0 THEN
			Q_sDiag 		:='Switch OFF Timer abgelaufen';
			act_Diag();
		END_IF
		IF I_stInfoData.nMapDiag.1 THEN
			Q_sDiag 		:='Switch ON Timer abgelaufen';
			act_Diag();
		END_IF
	END_CASE

	(* ========================================================= *)
	(*BE*)
END_ACTION

ACTION actInfoEStop:
	(* TwinSAFE-Funktionsbaustein FB EStop *)
	(* ========================================================= *)
	Q_bErrorState		:= FALSE;
	Q_bErrorDiag		:= FALSE;
	Q_sState			:= '';
	Q_sDiag				:= '';

	sFB				:= CONCAT('TwinSAFE Gruppe',INT_TO_STRING(I_nGrpId));
	sFB				:= CONCAT(sFB,' => ');
	sFB				:= CONCAT(sFB,'FB');
	sFB				:= CONCAT(sFB,INT_TO_STRING(I_nFBId));
	sFB				:= CONCAT(sFB,' ');
	sFB				:= CONCAT(sFB,I_sFBName);
	sFB				:= CONCAT(sFB,' => ');
	(* ========================================================= *)
	(* State *)
	CASE I_stInfoData.nMapState OF
		0:	Q_sState		:= 'undefiniert';
			act_State();

		1:	Q_sState		:= 'Run';

		2:	Q_sState		:= 'Stop';

		3:	Q_sState		:= 'Safe';

		4:	Q_sState		:= 'Error';
			act_State();

		5:	Q_sState		:= 'Reset';

		6:	Q_sState		:= 'Start';

		8:	Q_sState		:= 'DelayOut';

	ELSE	Q_sState		:= 'Error';
			act_State();
	END_CASE

	(* ========================================================= *)
	(* Diagnose *)
	CASE I_stInfoData.nMapDiag OF
		0: Q_sDiag :='-';
	ELSE
		IF I_stInfoData.nMapDiag.0 THEN
			Q_sDiag 			:='Diskrepanz Fehler Eingangsgruppe 1 => Safety Input => ';
			Q_sDiag				:= CONCAT(Q_sDiag,I_sNameEinGruppe1);
			act_Diag();
		END_IF

		IF I_stInfoData.nMapDiag.1 THEN
			Q_sDiag 			:='Diskrepanz Fehler Eingangsgruppe 2 => Safety Input => ';
			Q_sDiag				:= CONCAT(Q_sDiag,I_sNameEinGruppe2);
			act_Diag();
		END_IF

		IF I_stInfoData.nMapDiag.2 THEN
			Q_sDiag 			:='Diskrepanz Fehler Eingangsgruppe 3 => Safety Input => ';
			Q_sDiag				:= CONCAT(Q_sDiag,I_sNameEinGruppe3);
			act_Diag();
		END_IF

		IF I_stInfoData.nMapDiag.3 THEN
			Q_sDiag 			:='Diskrepanz Fehler Eingangsgruppe 4 => Safety Input => ';
			Q_sDiag				:= CONCAT(Q_sDiag,I_sNameEinGruppe4);
			act_Diag();
		END_IF

		IF I_stInfoData.nMapDiag.4 THEN
			Q_sDiag 			:='Rueckfuehrkreis Fehler EDM1 => Safety Input => ';
			Q_sDiag				:= CONCAT(Q_sDiag,I_sNameEMD1);
			act_Diag();
		END_IF

		IF I_stInfoData.nMapDiag.5 THEN
			Q_sDiag 			:='Rueckfuehrkreis Fehler EDM2 => Safety Input => ';
			Q_sDiag				:= CONCAT(Q_sDiag,I_sNameEMD2);
			act_Diag();
		END_IF
	END_CASE

	(* ========================================================= *)
	(*BE*)
END_ACTION

ACTION actInfoMON:
	(* TwinSAFE-Funktionsbaustein FB MOM *)
	(* ========================================================= *)
	Q_bErrorState		:= FALSE;
	Q_bErrorDiag		:= FALSE;
	Q_sState			:= '';
	Q_sDiag				:= '';

	sFB				:= CONCAT('TwinSAFE Gruppe',INT_TO_STRING(I_nGrpId));
	sFB				:= CONCAT(sFB,' => ');
	sFB				:= CONCAT(sFB,'FB');
	sFB				:= CONCAT(sFB,INT_TO_STRING(I_nFBId));
	sFB				:= CONCAT(sFB,' ');
	sFB				:= CONCAT(sFB,I_sFBName);
	sFB				:= CONCAT(sFB,' => ');

	(* ========================================================= *)
	(* State *)
	CASE I_stInfoData.nMapState OF
		0:	Q_sState		:= 'undefiniert';
			act_State();

		1:	Q_sState		:= 'Run';

		2:	Q_sState		:= 'Stop';

		3:	Q_sState		:= 'Safe';

		4:	Q_sState		:= 'Error';
			act_State();

		5:	Q_sState		:= 'Reset';

		6:	Q_sState		:= 'Start';

		7:	Q_sState		:= 'ErrorDelay';
			act_State();

		8:	Q_sState		:= 'DelayOut';

		9:	Q_sState		:= 'FuncTest';

	ELSE	Q_sState		:= 'Error';
			act_State();
	END_CASE

	(* ========================================================= *)
	(* Diagnose *)
	CASE I_stInfoData.nMapDiag OF
		0: ;
	ELSE
		IF I_stInfoData.nMapDiag.0 THEN
			Q_sDiag 			:='Diskrepanz Fehler Eingangsgruppe 1 => Safety Input => ';
			Q_sDiag				:= CONCAT(Q_sDiag,I_sNameEinGruppe1);
			act_Diag();
		END_IF

		IF I_stInfoData.nMapDiag.1 THEN
			Q_sDiag 			:='Diskrepanz Fehler Eingangsgruppe 2 => Safety Input => ';
			Q_sDiag				:= CONCAT(Q_sDiag,I_sNameEinGruppe2);
			act_Diag();
		END_IF

		IF I_stInfoData.nMapDiag.2 THEN
			Q_sDiag 			:='Diskrepanz Fehler Secure-Eingangsgruppe => Safety Input => ';
			Q_sDiag				:= CONCAT(Q_sDiag,I_sNameSecGruppe);
			act_Diag();
		END_IF

		IF I_stInfoData.nMapDiag.4 THEN
			Q_sDiag 			:='Rueckfuehrkreis Fehler EDM1 => Safety Input => ';
			Q_sDiag				:= CONCAT(Q_sDiag,I_sNameEMD1);
			act_Diag();
		END_IF

		IF I_stInfoData.nMapDiag.5 THEN
			Q_sDiag 			:='Rueckfuehrkreis Fehler EDM2 => Safety Input => ';
			Q_sDiag				:= CONCAT(Q_sDiag,I_sNameEMD2);
			act_Diag();
		END_IF
	END_CASE

	(* ========================================================= *)
	(*BE*)
END_ACTION

ACTION actInfoMuting:
	(* TwinSAFE-Funktionsbaustein FB MUTING*)
	(* ========================================================= *)
	Q_bErrorState		:= FALSE;
	Q_bErrorDiag		:= FALSE;
	Q_sState			:= '';
	Q_sDiag				:= '';

	sFB				:= CONCAT('TwinSAFE Gruppe',INT_TO_STRING(I_nGrpId));
	sFB				:= CONCAT(sFB,' => ');
	sFB				:= CONCAT(sFB,'FB');
	sFB				:= CONCAT(sFB,INT_TO_STRING(I_nFBId));
	sFB				:= CONCAT(sFB,' ');
	sFB				:= CONCAT(sFB,I_sFBName);
	sFB				:= CONCAT(sFB,' => ');

	(* ========================================================= *)
	(* State *)
	CASE I_stInfoData.nMapState OF
		0:	Q_sState		:= 'undefiniert';
			act_State();

		1:	Q_sState		:= 'Run';

		2:	Q_sState		:= 'Stop';

		4:	Q_sState		:= 'Safe';

		5:	Q_sState		:= 'Reset';

		6:	Q_sState		:= 'undefiniert';
			act_State();

		7:	Q_sState		:= 'undefiniert';
			act_State();

		8:	Q_sState		:= 'DelayOut';

		9:	Q_sState		:= 'Muting1';
		10:Q_sState		:= 'Muting2';
		11:Q_sState		:= 'Muting3';
		12:Q_sState		:= 'Muting4';
		13:Q_sState		:= 'Muting5';
		14:Q_sState		:= 'Muting6';
		15:Q_sState		:= 'Muting7';
		16:Q_sState		:= 'Muting8';
		17:Q_sState		:= 'Muting9';

	ELSE 	Q_sState		:= 'Error';
			act_State();
	END_CASE

	(* ========================================================= *)
	(* Diagnose *)
	CASE I_stInfoData.nMapDiag OF
		0: ;
	ELSE
		IF I_stInfoData.nMapDiag.0 THEN
			Q_sDiag 			:='Diskrepanz Fehler Muting Eingangsgruppe 1 => Safety Input => ';
			Q_sDiag				:= CONCAT(Q_sDiag,I_sNameEinGruppe1);
			act_Diag();
		END_IF

		IF I_stInfoData.nMapDiag.1 THEN
			Q_sDiag 			:='Diskrepanz Fehler OSSD Eingangsgruppe => Safety Input => ';
			Q_sDiag				:= CONCAT(Q_sDiag,I_sNameOSSDEinGruppe);
			act_Diag();
		END_IF

		IF I_stInfoData.nMapDiag.2 THEN
			Q_sDiag 			:='Diskrepanz Fehler Muting Eingangsgruppe 2 => Safety Input => ';
			Q_sDiag				:= CONCAT(Q_sDiag,I_sNameEinGruppe2);
			act_Diag();
		END_IF

		IF I_stInfoData.nMapDiag.4 THEN
			Q_sDiag 			:='Rueckfuehrkreis Fehler EDM1 => Safety Input => ';
			Q_sDiag				:= CONCAT(Q_sDiag,I_sNameEMD1);
			act_Diag();
		END_IF

		IF I_stInfoData.nMapDiag.5 THEN
			Q_sDiag 			:='Rueckfuehrkreis Fehler EDM2 => Safety Input => ';
			Q_sDiag				:= CONCAT(Q_sDiag,I_sNameEMD2);
			act_Diag();
		END_IF

		IF I_stInfoData.nMapDiag.6 THEN
			Q_sDiag 			:='Mutingsequenz wurde verletzt';
			act_Diag();
		END_IF

		IF I_stInfoData.nMapDiag.7 THEN
			Q_sDiag 			:='Maximale Mutingtime wurde überschritten';
			act_Diag();
		END_IF
	END_CASE

	(* ========================================================= *)
	(*BE*)
END_ACTION

ACTION actInfoOPMode:
	(* TwinSAFE-Funktionsbaustein FB OPMode *)
	(* ========================================================= *)
	Q_bErrorState		:= FALSE;
	Q_bErrorDiag		:= FALSE;
	Q_sState			:= '';
	Q_sDiag				:= '';

	sFB				:= CONCAT('TwinSAFE Gruppe',INT_TO_STRING(I_nGrpId));
	sFB				:= CONCAT(sFB,' => ');
	sFB				:= CONCAT(sFB,'FB');
	sFB				:= CONCAT(sFB,INT_TO_STRING(I_nFBId));
	sFB				:= CONCAT(sFB,' ');
	sFB				:= CONCAT(sFB,I_sFBName);
	sFB				:= CONCAT(sFB,' => ');

	(* ========================================================= *)
	(* State *)
	CASE I_stInfoData.nMapState OF
		0:	Q_sState		:= 'undefiniert';
			act_State();

		1:	Q_sState		:= 'Run';

		2:	Q_sState		:= 'Stop';

		3:	Q_sState		:= 'Safe';

		4:	Q_sState		:= 'ERROR';
			act_State();

		5:	Q_sState		:= 'Reset';

		6:	Q_sState		:= 'Start';

	ELSE	Q_sState		:= 'Error';
			act_State();
	END_CASE

	(* ========================================================= *)
	(* Diagnose *)
	(*	stInfoData.uiMapDiag	immer gleich 0*)
	CASE I_stInfoData.nMapState OF
		0: ;
	ELSE
		IF I_stInfoData.nMapDiag.0 THEN
			Q_sDiag 		:= 'Diskrepanzueberwachungsfehler';
			act_Diag();
		END_IF
	END_CASE

	(* ========================================================= *)
	(*BE*)
END_ACTION

ACTION actInfoOR:
	(* TwinSAFE-Funktionsbaustein FB OR *)
	(* ========================================================= *)
	Q_bErrorState		:= FALSE;
	Q_bErrorDiag		:= FALSE;
	Q_sState			:= '';
	Q_sDiag				:= '';

	sFB				:= CONCAT('TwinSAFE Gruppe',INT_TO_STRING(I_nGrpId));
	sFB				:= CONCAT(sFB,' => ');
	sFB				:= CONCAT(sFB,'FB');
	sFB				:= CONCAT(sFB,INT_TO_STRING(I_nFBId));
	sFB				:= CONCAT(sFB,' ');
	sFB				:= CONCAT(sFB,I_sFBName);
	sFB				:= CONCAT(sFB,' => ');

	(* ========================================================= *)
	(* State *)
	CASE I_stInfoData.nMapState OF
		0:	Q_sState		:= 'undefiniert';
			act_State();

		1:	Q_sState		:= 'Run';

		2:	Q_sState		:= 'Stop';

		3:	Q_sState		:= 'Safe';

	ELSE	Q_sState		:= 'ERROR';
			act_State();
	END_CASE

	(* ========================================================= *)
	(* Diagnose *)
	(*	stInfoData.uiMapDiag	immer gleich 0*)
	CASE I_stInfoData.nMapState OF
		0:	;
	END_CASE

	(* ========================================================= *)
	(*BE*)
END_ACTION

ACTION actInfoRS:
	(* TwinSAFE-Funktionsbaustein FB RS *)
	(* ========================================================= *)
	Q_bErrorState		:= FALSE;
	Q_bErrorDiag		:= FALSE;
	Q_sState			:= '';
	Q_sDiag				:= '';

	sFB				:= CONCAT('TwinSAFE Gruppe',INT_TO_STRING(I_nGrpId));
	sFB				:= CONCAT(sFB,' => ');
	sFB				:= CONCAT(sFB,'FB');
	sFB				:= CONCAT(sFB,INT_TO_STRING(I_nFBId));
	sFB				:= CONCAT(sFB,' ');
	sFB				:= CONCAT(sFB,I_sFBName);
	sFB				:= CONCAT(sFB,' => ');

	(* ========================================================= *)
	(* State *)
	CASE I_stInfoData.nMapState OF
		0:	Q_sState		:= 'undefiniert';
			act_State();

		2:	Q_sState		:= 'Stop';

		3:	Q_sState		:= 'Safe';

		9:	Q_sState		:= 'Set';

	ELSE	Q_sState		:= 'Error';
			act_State();
	END_CASE

	(* ========================================================= *)
	(* Diagnose *)
	(*	stInfoData.uiMapDiag	immer gleich 0*)
	CASE I_stInfoData.nMapState OF
		0:	;
	END_CASE

	(* ========================================================= *)
	(*BE*)
END_ACTION

ACTION actInfoSR:
	(* TwinSAFE-Funktionsbaustein FB SR *)
	(* ========================================================= *)
	Q_bErrorState		:= FALSE;
	Q_bErrorDiag		:= FALSE;
	Q_sState			:= '';
	Q_sDiag				:= '';

	sFB				:= CONCAT('TwinSAFE Gruppe',INT_TO_STRING(I_nGrpId));
	sFB				:= CONCAT(sFB,' => ');
	sFB				:= CONCAT(sFB,'FB');
	sFB				:= CONCAT(sFB,INT_TO_STRING(I_nFBId));
	sFB				:= CONCAT(sFB,' ');
	sFB				:= CONCAT(sFB,I_sFBName);
	sFB				:= CONCAT(sFB,' => ');

	(* ========================================================= *)
	(* State *)
	CASE I_stInfoData.nMapState OF
		0:	Q_sState		:= 'undefiniert';
			act_State();

		2:	Q_sState		:= 'Stop';

		3:	Q_sState		:= 'Safe';

		9:	Q_sState		:= 'Set';

	ELSE	Q_sState		:= 'Error';
			act_State();
	END_CASE

	(* ========================================================= *)
	(* Diagnose *)
	(*	stInfoData.uiMapDiag	immer gleich 0*)
	CASE I_stInfoData.nMapState OF
		0:	;
	END_CASE

	(* ========================================================= *)
	(*BE*)
END_ACTION

ACTION actInfoTOF:
	(* TwinSAFE-Funktionsbaustein FB TON *)
	(* ========================================================= *)
	Q_bErrorState		:= FALSE;
	Q_bErrorDiag		:= FALSE;
	Q_sState			:= '';
	Q_sDiag				:= '';

	sFB				:= CONCAT('TwinSAFE Gruppe',INT_TO_STRING(I_nGrpId));
	sFB				:= CONCAT(sFB,' => ');
	sFB				:= CONCAT(sFB,'FB');
	sFB				:= CONCAT(sFB,INT_TO_STRING(I_nFBId));
	sFB				:= CONCAT(sFB,' ');
	sFB				:= CONCAT(sFB,I_sFBName);
	sFB				:= CONCAT(sFB,' => ');

	(* ========================================================= *)
	(* State *)
	CASE I_stInfoData.nMapState OF
		0:	Q_sState		:= 'undefiniert';
			act_State();

		1:	Q_sState		:= 'Run';

		2:	Q_sState		:= 'Stop';

		3:	Q_sState		:= 'Safe';

		9:	Q_sState		:= 'Delay_Out';

	ELSE	Q_sState		:= 'Error';
			act_State();
	END_CASE

	(* ========================================================= *)
	(* Diagnose *)
	(*	stInfoData.uiMapDiag	immer gleich 0*)
	CASE I_stInfoData.nMapState OF
		0:	;
	END_CASE

	(* ========================================================= *)
	(*BE*)
END_ACTION

ACTION actInfoTON:
	(* TwinSAFE-Funktionsbaustein FB TON *)
	(* ========================================================= *)
	Q_bErrorState		:= FALSE;
	Q_bErrorDiag		:= FALSE;
	Q_sState			:= '';
	Q_sDiag				:= '';

	sFB				:= CONCAT('TwinSAFE Gruppe',INT_TO_STRING(I_nGrpId));
	sFB				:= CONCAT(sFB,' => ');
	sFB				:= CONCAT(sFB,'FB');
	sFB				:= CONCAT(sFB,INT_TO_STRING(I_nFBId));
	sFB				:= CONCAT(sFB,' ');
	sFB				:= CONCAT(sFB,I_sFBName);
	sFB				:= CONCAT(sFB,' => ');

	(* ========================================================= *)
	(* State *)
	CASE I_stInfoData.nMapState OF
		0:	Q_sState		:= 'undefiniert';
			act_State();

		1:	Q_sState		:= 'Run';

		2:	Q_sState		:= 'Stop';

		3:	Q_sState		:= 'Safe';

		9:	Q_sState		:= 'Delay_In';

	ELSE	Q_sState		:= 'Error';
			act_State();
	END_CASE

	(* ========================================================= *)
	(* Diagnose *)
	(*	stInfoData.uiMapDiag	immer gleich 0*)
	CASE I_stInfoData.nMapState OF
		0:	;
	END_CASE

	(* ========================================================= *)
	(*BE*)
END_ACTION

ACTION actInfoTwoHand:
	(* TwinSAFE-Funktionsbaustein FB AND*)
	(* ========================================================= *)
	Q_bErrorState		:= FALSE;
	Q_bErrorDiag		:= FALSE;
	Q_sState			:= '';
	Q_sDiag				:= '';

	sFB				:= CONCAT('TwinSAFE Gruppe',INT_TO_STRING(I_nGrpId));
	sFB				:= CONCAT(sFB,' => ');
	sFB				:= CONCAT(sFB,'FB');
	sFB				:= CONCAT(sFB,INT_TO_STRING(I_nFBId));
	sFB				:= CONCAT(sFB,' ');
	sFB				:= CONCAT(sFB,I_sFBName);
	sFB				:= CONCAT(sFB,' => ');

	(* ========================================================= *)
	(* State *)
	CASE I_stInfoData.nMapState OF
		0:	Q_sState		:= 'undefiniert';
			act_State();

		1:	Q_sState		:= 'Run';

		2:	Q_sState		:= 'Stop';

		3:	Q_sState		:= 'Safe';

		4:	Q_sState		:= 'Error';
			act_State();

		5:	Q_sState		:= 'Reset';

		6:	Q_sState		:= 'Start';

		11:Q_sState		:= '1Button';

		12:Q_sState		:= '2Button';

		13:Q_sState		:= 'Release';

	ELSE	Q_sState		:= 'Error';
			act_State();
	END_CASE

	(* ========================================================= *)
	(* Diagnose *)
	CASE I_stInfoData.nMapDiag OF
		0: ;
	ELSE
		IF I_stInfoData.nMapDiag.0 THEN
			Q_sDiag 			:='Diskrepanz Fehler Eingangsgruppe 1 => Safety Input => ';
			Q_sDiag				:= CONCAT(Q_sDiag,I_sNameEinGruppe1);
			act_Diag();
		END_IF

		IF I_stInfoData.nMapDiag.1 THEN
			Q_sDiag 			:='Diskrepanz Fehler Eingangsgruppe 2 => Safety Input => ';
			Q_sDiag				:= CONCAT(Q_sDiag,I_sNameEinGruppe2);
			act_Diag();
		END_IF

		IF I_stInfoData.nMapDiag.2 THEN
			Q_sDiag 			:='Diskrepanz Fehler zwischen den beiden Eingangsgruppe => Safety Input => ';
			Q_sDiag				:= CONCAT(Q_sDiag,I_sNameEinGruppe1);
			Q_sDiag				:= CONCAT(Q_sDiag,'_');
			Q_sDiag				:= CONCAT(Q_sDiag,I_sNameEinGruppe2);
			act_Diag();
		END_IF
	END_CASE

	(* ========================================================= *)
	(*BE*)
END_ACTION

END_FUNCTION_BLOCK

// POUs/DiagSafety/FB_TwinSAFE_Group_Info
(* Version arrHistory: 
Description: Ethercat-Saftey Diagnose
Date          | Version    | created under        | Author          | Remark 
---------------------------------------------------------------------------------------- 
12/09/2011    | 1.1.0      | V2.11.0 (Build 1551) | T.Löhner        | first release
*)
FUNCTION_BLOCK FB_TwinSAFE_Group_Info
VAR_INPUT
	I_stInfoData	: ST_TwinSAFE_Group_Info;
	I_nGrpId			: INT;
END_VAR
VAR_OUTPUT
	Q_bErrorState	: BOOL;
	Q_sState			: STRING;
END_VAR
VAR
	sGrp				: STRING;
	sState_old		: Tc2_System.T_MaxString;
	tonStateChange	: TON;
END_VAR

	(* ========================================================= *)
		actInfo();
	(* ========================================================= *)

ACTION act_State:

	IF Q_sState<> sState_old THEN
		Q_bErrorState	:= FALSE;
	ELSE
		Q_bErrorState	:= TRUE;
	END_IF

	tonStateChange(
		IN:= NOT Q_bErrorState,
		PT:=t#500ms);

	IF tonStateChange.Q THEN
		sState_old	:= Q_sState;
	END_IF

	Q_sState		:= CONCAT('Status: ',Q_sState);
	Q_sState		:= CONCAT(sGrp,Q_sState);

	(*BE*)
END_ACTION

ACTION actInfo:
	(* TwinSAFE-Group *)
	(* ========================================================= *)
	Q_bErrorState			:= FALSE;
	Q_sState				:= '';

	sGrp					:= CONCAT('TwinSAFE Gruppe',INT_TO_STRING(I_nGrpId));
	sGrp					:= CONCAT(sGrp,' => ');

(* ========================================================= *)
	(* State *)
	CASE I_stInfoData.nMapState OF
		1: 	Q_sState 			:='Run';

		2: 	Q_sState 			:='Stop';

		3: 	Q_sState 			:='Safe';

		4: 	Q_sState 			:='Error';
				act_State();

		5: 	Q_sState 			:='Reset';

	ELSE		Q_sState 			:='undefiniert';
				act_State();
	END_CASE

	(* ========================================================= *)
END_ACTION

END_FUNCTION_BLOCK

// POUs/DiagSafety/FB_TwinSAFEConnInfo
(* Version History: 
Description: Ethercat-Saftey Diagnose für TwinSAFE-Verbindungen
Date			| Version	| created under			| Author				| Remark 
---------------------------------------------------------------------------------------- 
12/09/2011	| 1.1.0		| V2.11.0 (Build 1551)	| T.Löhner			| first release 
28.02.2023	| 1.2.0		| V3.1.4024.40				| B.Daut				| Adaptiert für Avalon-HMI Meldesystem
*)
FUNCTION_BLOCK FB_TwinSAFEConnInfo
VAR_IN_OUT
	IQ_stMeldung	: ST_MeldSafetyOuts;
END_VAR
VAR_INPUT
	I_stInfoData	: ST_TwinSAFE_Conn_Info;	// TwinSAFE-Connection zu einer Klemme bzw. Alias
	I_nGrpId			: INT;	// TwinSAFE-Gruppe zur Erstellung der Fehlermeldung
	I_nConnId		: INT;	// TwinSAFE-ConnectionID zur Erstellung der Fehlermeldung
	I_sConnName		: Tc2_System.T_MaxString;	// TwinSAFE-ConnectionName zur Erstellung der Fehlermeldung
	I_bMeldungFreigaben	: BOOL;	// TwinSAFE-Connection darf überwacht werden. z.B. bFehlerEtherCATAllg
END_VAR
VAR
	sConn				: STRING;
	nDiag				: INT;
	sState_old		: Tc2_System.T_MaxString;	// Zum feststellen einer Änderung und damit einhergehenden Neuauslösung der Meldung
	sDiag_old		: Tc2_System.T_MaxString;	// Zum feststellen einer Änderung und damit einhergehenden Neuauslösung der Meldung
	tonStateChange	: Tc2_Standard.TON;	// Zum feststellen einer Änderung und damit einhergehenden Neuauslösung der Meldung
	tonDiagChange	: Tc2_Standard.TON;	// Zum feststellen einer Änderung und damit einhergehenden Neuauslösung der Meldung
END_VAR

	(* ========================================================= *)
	actInfo();

	(* ========================================================= *)

ACTION act_Diag:

	IF IQ_stMeldung.sDiag<> sDiag_old THEN
		IQ_stMeldung.bMeldDiag	:= FALSE;
	ELSE
		IQ_stMeldung.bMeldDiag	:= I_bMeldungFreigaben;
	END_IF

	tonDiagChange(
		IN:= NOT IQ_stMeldung.bMeldDiag,
		PT:=t#500ms);

	IF tonDiagChange.Q THEN
		sDiag_old	:= IQ_stMeldung.sDiag;
	END_IF

	IQ_stMeldung.sDiag	:= CONCAT('Diagnose: ',IQ_stMeldung.sDiag);
	IQ_stMeldung.sDiag	:= CONCAT(sConn,IQ_stMeldung.sDiag);

	(*BE*)
END_ACTION

ACTION act_State:

	IF IQ_stMeldung.sState<> sState_old THEN
		IQ_stMeldung.bMeldState	:= FALSE;
	ELSE
		IQ_stMeldung.bMeldState	:= I_bMeldungFreigaben;
	END_IF

	tonStateChange(
		IN:= NOT IQ_stMeldung.bMeldState,
		PT:=t#500ms);

	IF tonStateChange.Q THEN
		sState_old	:= IQ_stMeldung.sState;
	END_IF

	IQ_stMeldung.sState	:= CONCAT('Status: ',IQ_stMeldung.sState);
	IQ_stMeldung.sState	:= CONCAT(sConn,IQ_stMeldung.sState);

	(*BE*)
END_ACTION

ACTION actInfo:
	(* TwinSAFE-Connection *)
	(* ========================================================= *)
	IQ_stMeldung.bMeldDiag	:= FALSE;
	IQ_stMeldung.bMeldState	:= FALSE;
	IQ_stMeldung.sDiag		:= '';
	IQ_stMeldung.sState		:= '';

	sConn				:= CONCAT('TwinSAFE Gruppe',INT_TO_STRING(I_nGrpId));
	sConn				:= CONCAT(sConn,' => ');
	sConn				:= CONCAT(sConn,'Connection');
	sConn				:= CONCAT(sConn,INT_TO_STRING(I_nConnId));
	sConn				:= CONCAT(sConn,' ');
	sConn				:= CONCAT(sConn,I_sConnName);
	sConn				:= CONCAT(sConn,' => ');

	(* ========================================================= *)
	(* State *)
	CASE I_stInfoData.nMapState OF
		100:	IQ_stMeldung.sState	:='Reset';

		101:	IQ_stMeldung.sState	:='Session';

		102:	IQ_stMeldung.sState	:='Connection';

		103:	IQ_stMeldung.sState	:='Parameter';

		104:	IQ_stMeldung.sState	:='Data';

		105:	IQ_stMeldung.sState	:='Shutdown';

	ELSE
		IQ_stMeldung.sState	:='undefiniert';
		act_State();
	END_CASE

	(* ========================================================= *)
	(* Diagnose *)
	CASE I_stInfoData.nMapDiag OF
			0: ;
	ELSE
		nDiag	:= WORD_TO_INT(UINT_TO_WORD(I_stInfoData.nMapDiag) AND 16#000F);
		CASE nDiag OF
			1: IQ_stMeldung.sDiag	:='Ungueltiges Kommando';
				act_Diag();

			2: IQ_stMeldung.sDiag	:='Unbekanntes Kommando';
				act_Diag();

			3: IQ_stMeldung.sDiag	:='Ungueltige Connection ID';
				act_Diag();

			4: IQ_stMeldung.sDiag	:='Ungueltige CRC';
				act_Diag();

			5: IQ_stMeldung.sDiag	:='Watchdog abgelaufen';
				act_Diag();

			6: IQ_stMeldung.sDiag	:='Ungueltige FSoE address';
				act_Diag();

			7: IQ_stMeldung.sDiag	:='Ungueltige data';
				act_Diag();

			8: IQ_stMeldung.sDiag	:='Ungueltige Kommunikationsparameterlaenge';
				act_Diag();

			9: IQ_stMeldung.sDiag	:='Ungueltige Kommunikationsparameter';
				act_Diag();

			10:IQ_stMeldung.sDiag	:='Ungueltige Anwenderparameterlaenge';
				act_Diag();

			11:IQ_stMeldung.sDiag	:='Ungueltige Anwenderparameter';
				act_Diag();

			12:IQ_stMeldung.sDiag	:='FSoE Master Reset';
				act_Diag();
		END_CASE

		nDiag:=WORD_TO_INT(UINT_TO_WORD(I_stInfoData.nMapDiag) AND 16#00F0);
		nDiag:=SHL(nDiag,4);
		CASE nDiag OF
			1 :IQ_stMeldung.sDiag	:='Fehler beim FSoE erkannt';
				act_Diag();

			2 :IQ_stMeldung.sDiag	:='FSoE Slave meldet Failsafe Value aktiv';
				act_Diag();

			4 :IQ_stMeldung.sDiag	:='StartUp';
				act_Diag();

			8 :IQ_stMeldung.sDiag	:='FSoE Master meldet Failsafe Value akriv';
				act_Diag();
		END_CASE
	END_CASE

	(* ========================================================= *)
END_ACTION

END_FUNCTION_BLOCK

// POUs/DiagSafety/FB_TwinSAFEConnInfo4Byte
(* Version history:
Description: Ethercat-Saftey Diagnose
Date          | Version    | created under        | Author          | Remark 
---------------------------------------------------------------------------------------- 
12/09/2011    | 1.1.0      | V2.11.0 (Build 1551) | T.Löhner        | first release
25/04/2018    | 1.1.1      | V2.11.0 (Build 4022) | B.Daut	        | bugfix und weitere Fehlermeldung hinzugefügt
*)
FUNCTION_BLOCK FB_TwinSAFEConnInfo4Byte
VAR_OUTPUT
	Q_bErrorDiag	: BOOL;
	Q_bErrorState	: BOOL;
	Q_sDiag			: Tc2_System.T_MaxString;
	Q_sState			: Tc2_System.T_MaxString;
	Q_sState2		: Tc2_System.T_MaxString;
END_VAR

VAR_INPUT
	I_stInfoData	: ST_TwinSAFEConnInfo4Byte;
	I_nGrpId			: INT	:= 1;
	I_bGroupDeaktivated	: BOOL;	// Wenn die TwinSAFE-Gruppe deaktiviert wurde, darf die Connection kein Meldung absetzen
	I_nConnId		: INT;
	I_sConnName		: Tc2_System.T_MaxString;
END_VAR
VAR
	sConn				: Tc2_System.T_MaxString;
	nDiag				: WORD;
	sStateOld		: Tc2_System.T_MaxString;
	sDiagOld			: Tc2_System.T_MaxString;
	tonStateChange	: Tc2_Standard.TON;
	tonDiagChange	: Tc2_Standard.TON;
END_VAR

//****************************************************************************************************
a_Info();

//****************************************************************************************************
// ENDE

ACTION a_Info:
// TwinSAFE-Connection
//****************************************************************************************************
Q_bErrorState		:= FALSE;
Q_bErrorDiag		:= FALSE;
Q_sState				:= '';
Q_sState2			:= '';
Q_sDiag				:= '';

sConn				:= CONCAT('Gruppe',INT_TO_STRING(I_nGrpId));
sConn				:= CONCAT(sConn,' => ');
sConn				:= CONCAT(sConn,'Connection');
sConn				:= CONCAT(sConn,INT_TO_STRING(I_nConnId));
sConn				:= CONCAT(sConn,' ');
sConn				:= CONCAT(sConn,I_sConnName);
sConn				:= CONCAT(sConn,' => ');

//****************************************************************************************************
// Klartext aus der Doku zur EL6900 PDF, Seite 16 oben, Tabelle 2-5

// State
CASE I_stInfoData.nMapState
OF

100: 	Q_sState 			:='Reset';
		Q_sState2			:='Der Zustand Reset dient dazu, nach dem Power-On oder einem Safety over EtherCAT Kommunikationsfehler die Safety over EtherCAT Connection neu zu initialisieren.';

101: 	Q_sState 			:='Session';
		Q_sState2			:='Beim Übergang in den bzw. im Zustand Session wird eine Session ID vom Safety over EtherCAT Master zum Safety over EtherCAT Slave übertragen, der wiederum mit einer eigenen Session ID antwortet.';

102: 	Q_sState 			:='Connection';
		Q_sState2			:='Im Zustand Connection wird eine Connection ID vom Safety over EtherCAT Master zum Safety over EtherCAT Slave übertragen.';

103: 	Q_sState 			:='Parameter';
		Q_sState2			:='Im Zustand Parameter werden sichere Kommunikations- und gerätespezifische Anwendungsparameter übertragen.';

104: 	Q_sState 			:='Data';
		Q_sState2			:='Im Zustand Data werden solange Safety over EtherCAT Cycles übertragen, bis entweder ein Kommunikationsfehler auftritt oder ein Safety over EtherCAT Node lokal gestoppt wird.';

105: 	Q_sState 			:='Shutdown';
		Q_sState2			:='Im Zustand Shutdown ist die Verbindung durch einen der Kommunikationspartner heruntergefahren worden.';

ELSE
	Q_sState 			:='undefiniert';
	Q_sState2			:='';
	b_State();
END_CASE

//****************************************************************************************************
// Klartext aus der Doku zur EL6900 PDF, Seite 15 unten, Tabelle 2-4

// Diagnose

// Die Fehlerbits 0-3 kommen parallel, können also als Zahlen abgefragt werden
CASE I_stInfoData.nMapDiag OF
		0: ;
ELSE
	nDiag	:=UINT_TO_WORD(I_stInfoData.nMapDiag) AND 16#000F;
	CASE nDiag OF
		1: Q_sDiag			:='Ungueltiges Kommando';
			c_Diag();

		2: Q_sDiag 			:='Unbekanntes Kommando';
			c_Diag();

		3: Q_sDiag 			:='Ungueltige Connection ID';
			c_Diag();

		4: Q_sDiag 			:='Ungueltige CRC';
			c_Diag();

		5: Q_sDiag 			:='Watchdog abgelaufen';
			c_Diag();

		6: Q_sDiag 			:='Ungueltige FSoE address';
			c_Diag();

		7: Q_sDiag 			:='Ungueltige data';
			c_Diag();

		8: Q_sDiag 			:='Ungueltige Kommunikationsparameterlaenge';
			c_Diag();

		9: Q_sDiag 			:='Ungueltige Kommunikationsparameter';
			c_Diag();

		10:Q_sDiag 			:='Ungueltige Anwenderparameterlaenge';
			c_Diag();

		11:Q_sDiag 			:='Ungueltige Anwenderparameter';
			c_Diag();

		12:Q_sDiag		 		:='FSoE Master Reset';
			c_Diag();

		13:Q_sDiag		 		:='Modulfehler auf Slave erkannt, bei aktivierter "Option Modulfehler" ist ComError';
			c_Diag();

		14:Q_sDiag		 		:='Modulfehler auf EL290x erkannt, bei aktivierter Option "Error acknowledge active"';
			c_Diag();

		15:Q_sDiag		 		:='Slave noch nicht gestartet, oder unerwartetes Fehlerargument';
			c_Diag();
	END_CASE

// Die Fehlerbits 4-7 kommen einzeln und müssen daher auch einzeln abgefragt werden.
	nDiag	:=UINT_TO_WORD(I_stInfoData.nMapDiag) AND 16#00F0;

	IF nDiag.4
	THEN
		Q_sDiag	:= 'Fehler beim FSoE Slave erkannt';
		c_Diag();
	ELSIF nDiag.5
	THEN
		Q_sDiag	:='FSoE Slave meldet Failsafe Value aktiv';
		c_Diag();
	ELSIF nDiag.6
	THEN
		Q_sDiag	:='StartUp';
		c_Diag();
	ELSIF nDiag.7
	THEN
		Q_sDiag	:='FSoE Master meldet Failsafe Value aktiv';
		c_Diag();
	END_IF

END_CASE

//****************************************************************************************************
// ENDE
END_ACTION

ACTION b_State:
//****************************************************************************************************
// Stateänderungen feststellen
IF Q_sState<> sStateOld
	OR I_bGroupDeaktivated
THEN
	Q_bErrorState	:= FALSE;
ELSE
	Q_bErrorState	:= TRUE;
END_IF

tonStateChange(
	IN	:= NOT Q_bErrorState,
	PT	:= T#500MS
);

IF tonStateChange.Q
THEN
	sStateOld	:= Q_sState;
END_IF

Q_sState	:= CONCAT('Status: ',Q_sState);
Q_sState	:= CONCAT(sConn,Q_sState);

//****************************************************************************************************
// ENDE
END_ACTION

ACTION c_Diag:
//****************************************************************************************************
// Diagänderungen feststellen
IF Q_sDiag<> sDiagOld
THEN
	Q_bErrorDiag	:= FALSE;
ELSE
	Q_bErrorDiag	:= TRUE;
END_IF

tonDiagChange(
	IN	:= NOT Q_bErrorDiag,
	PT	:= T#500MS
);

IF tonDiagChange.Q
THEN
	sDiagOld	:= Q_sDiag;
END_IF

Q_sDiag	:= CONCAT('Diagnose: ',Q_sDiag);
Q_sDiag	:= CONCAT(sConn,Q_sDiag);

//****************************************************************************************************
// ENDE
END_ACTION

END_FUNCTION_BLOCK

// POUs/DiagSafety/FB_TwinSAFEConnInfo4Byte_1
(* Version history:
Description: Ethercat-Saftey Diagnose
Date			| Version	| created under			| Author          | Remark 
---------------------------------------------------------------------------------------- 
12/09/2011	| 1.1.0		| V2.11.0 (Build 1551)	| T.Löhner        | first release
25/04/2018	| 1.1.1		| V2.11.0 (Build 4022)	| B.Daut				| bugfix und weitere Fehlermeldung hinzugefügt
28.02.2023	| 2.1.0		| V3.1.4024.40				| B.Daut				| Adaptiert für Avalon-HMI Meldesystem
*)
FUNCTION_BLOCK FB_TwinSAFEConnInfo4Byte_1
VAR_IN_OUT
	IQ_stMeldung			: ST_MeldSafetyOuts;
END_VAR
VAR_INPUT
	I_stInfoData			: ST_TwinSAFEConnInfo4Byte;
	I_nGrpId					: INT	:= 1;	// TwinSAFE-Gruppe zur Erstellung der Fehlermeldung
	I_bGroupDeaktivated	: BOOL;	// Wenn die TwinSAFE-Gruppe deaktiviert wurde, darf die Connection kein Meldung absetzen
	I_nConnId				: INT;	// TwinSAFE-ConnectionID zur Erstellung der Fehlermeldung
	I_sConnName				: Tc2_System.T_MaxString;	// TwinSAFE-ConnectionName zur Erstellung der Fehlermeldung
END_VAR
VAR
	sConn						: Tc2_System.T_MaxString;
	nDiag						: WORD;
	sStateOld				: Tc2_System.T_MaxString;	// Zum feststellen einer Änderung und damit einhergehenden Neuauslösung der Meldung
	sDiagOld					: Tc2_System.T_MaxString;	// Zum feststellen einer Änderung und damit einhergehenden Neuauslösung der Meldung
	tonStateChange			: Tc2_Standard.TON;	// Zum feststellen einer Änderung und damit einhergehenden Neuauslösung der Meldung
	tonDiagChange			: Tc2_Standard.TON;	// Zum feststellen einer Änderung und damit einhergehenden Neuauslösung der Meldung
END_VAR

//****************************************************************************************************
a_Info();

//****************************************************************************************************
// ENDE

ACTION a_Info:
// TwinSAFE-Connection
//****************************************************************************************************
IQ_stMeldung.bMeldState	:= FALSE;
IQ_stMeldung.bMeldDiag	:= FALSE;
IQ_stMeldung.sState		:= '';
IQ_stMeldung.sDiag		:= '';

sConn				:= CONCAT('Gruppe',INT_TO_STRING(I_nGrpId));
sConn				:= CONCAT(sConn,' => ');
sConn				:= CONCAT(sConn,'Connection');
sConn				:= CONCAT(sConn,INT_TO_STRING(I_nConnId));
sConn				:= CONCAT(sConn,' ');
sConn				:= CONCAT(sConn,I_sConnName);
sConn				:= CONCAT(sConn,' => ');

//****************************************************************************************************
// Klartext aus der Doku zur EL6900 PDF, Seite 16 oben, Tabelle 2-5

// State
CASE I_stInfoData.nMapState
OF

100: 	IQ_stMeldung.sState	:='Reset';
		IQ_stMeldung.sState	:=CONCAT (IQ_stMeldung.sState,'Der Zustand Reset dient dazu, nach dem Power-On oder einem Safety over EtherCAT Kommunikationsfehler die Safety over EtherCAT Connection neu zu initialisieren.');

101: 	IQ_stMeldung.sState	:='Session';
		IQ_stMeldung.sState	:=CONCAT (IQ_stMeldung.sState,'Beim Übergang in den bzw. im Zustand Session wird eine Session ID vom Safety over EtherCAT Master zum Safety over EtherCAT Slave übertragen, der wiederum mit einer eigenen Session ID antwortet.');

102: 	IQ_stMeldung.sState	:='Connection';
		IQ_stMeldung.sState	:=CONCAT (IQ_stMeldung.sState,'Im Zustand Connection wird eine Connection ID vom Safety over EtherCAT Master zum Safety over EtherCAT Slave übertragen.');

103: 	IQ_stMeldung.sState	:='Parameter';
		IQ_stMeldung.sState	:=CONCAT (IQ_stMeldung.sState,'Im Zustand Parameter werden sichere Kommunikations- und gerätespezifische Anwendungsparameter übertragen.');

104: 	IQ_stMeldung.sState	:='Data';
		IQ_stMeldung.sState	:=CONCAT (IQ_stMeldung.sState,'Im Zustand Data werden solange Safety over EtherCAT Cycles übertragen, bis entweder ein Kommunikationsfehler auftritt oder ein Safety over EtherCAT Node lokal gestoppt wird.');

105: 	IQ_stMeldung.sState	:='Shutdown';
		IQ_stMeldung.sState	:=CONCAT (IQ_stMeldung.sState,'Im Zustand Shutdown ist die Verbindung durch einen der Kommunikationspartner heruntergefahren worden.');

ELSE
	IQ_stMeldung.sState	:='undefiniert';
	IQ_stMeldung.sState	:='';
	b_State();
END_CASE

//****************************************************************************************************
// Klartext aus der Doku zur EL6900 PDF, Seite 15 unten, Tabelle 2-4

// Diagnose

// Die Fehlerbits 0-3 kommen parallel, können also als Zahlen abgefragt werden
CASE I_stInfoData.nMapDiag OF
		0: ;
ELSE
	nDiag	:=UINT_TO_WORD(I_stInfoData.nMapDiag) AND 16#000F;
	CASE nDiag OF
		1: IQ_stMeldung.sDiag	:='Ungueltiges Kommando';
			c_Diag();

		2: IQ_stMeldung.sDiag	:='Unbekanntes Kommando';
			c_Diag();

		3: IQ_stMeldung.sDiag	:='Ungueltige Connection ID';
			c_Diag();

		4: IQ_stMeldung.sDiag	:='Ungueltige CRC';
			c_Diag();

		5: IQ_stMeldung.sDiag	:='Watchdog abgelaufen';
			c_Diag();

		6: IQ_stMeldung.sDiag	:='Ungueltige FSoE address';
			c_Diag();

		7: IQ_stMeldung.sDiag	:='Ungueltige data';
			c_Diag();

		8: IQ_stMeldung.sDiag	:='Ungueltige Kommunikationsparameterlaenge';
			c_Diag();

		9: IQ_stMeldung.sDiag	:='Ungueltige Kommunikationsparameter';
			c_Diag();

		10:IQ_stMeldung.sDiag	:='Ungueltige Anwenderparameterlaenge';
			c_Diag();

		11:IQ_stMeldung.sDiag	:='Ungueltige Anwenderparameter';
			c_Diag();

		12:IQ_stMeldung.sDiag	:='FSoE Master Reset';
			c_Diag();

		13:IQ_stMeldung.sDiag	:='Modulfehler auf Slave erkannt, bei aktivierter "Option Modulfehler" ist ComError';
			c_Diag();

		14:IQ_stMeldung.sDiag	:='Modulfehler auf EL290x erkannt, bei aktivierter Option "Error acknowledge active"';
			c_Diag();

		15:IQ_stMeldung.sDiag	:='Slave noch nicht gestartet, oder unerwartetes Fehlerargument';
			c_Diag();
	END_CASE

// Die Fehlerbits 4-7 kommen einzeln und müssen daher auch einzeln abgefragt werden.
	nDiag	:=UINT_TO_WORD(I_stInfoData.nMapDiag) AND 16#00F0;

	IF nDiag.4
	THEN
		IQ_stMeldung.sDiag	:= 'Fehler beim FSoE Slave erkannt';
		c_Diag();
	ELSIF nDiag.5
	THEN
		IQ_stMeldung.sDiag	:='FSoE Slave meldet Failsafe Value aktiv';
		c_Diag();
	ELSIF nDiag.6
	THEN
		IQ_stMeldung.sDiag	:='StartUp';
		c_Diag();
	ELSIF nDiag.7
	THEN
		IQ_stMeldung.sDiag	:='FSoE Master meldet Failsafe Value aktiv';
		c_Diag();
	END_IF

END_CASE

//****************************************************************************************************
// ENDE
END_ACTION

ACTION b_State:
//****************************************************************************************************
// Stateänderungen feststellen
IF IQ_stMeldung.sState<> sStateOld
THEN
	IQ_stMeldung.bMeldState	:= FALSE;
ELSE
	IQ_stMeldung.bMeldState	:= NOT I_bGroupDeaktivated;
END_IF

tonStateChange(
	IN	:= NOT IQ_stMeldung.bMeldState,
	PT	:= T#500MS
);

IF tonStateChange.Q
THEN
	sStateOld	:= IQ_stMeldung.sState;
END_IF

IQ_stMeldung.sState	:= CONCAT('Status: ',IQ_stMeldung.sState);
IQ_stMeldung.sState	:= CONCAT(sConn,IQ_stMeldung.sState);

//****************************************************************************************************
// ENDE
END_ACTION

ACTION c_Diag:
//****************************************************************************************************
// Diagänderungen feststellen
IF IQ_stMeldung.sDiag<> sDiagOld
THEN
	IQ_stMeldung.bMeldDiag	:= FALSE;
ELSE
	IQ_stMeldung.bMeldDiag	:= NOT I_bGroupDeaktivated;
END_IF

tonDiagChange(
	IN	:= NOT IQ_stMeldung.bMeldDiag,
	PT	:= T#500MS
);

IF tonDiagChange.Q
THEN
	sDiagOld	:= IQ_stMeldung.sDiag;
END_IF

IQ_stMeldung.sDiag	:= CONCAT('Diagnose: ',IQ_stMeldung.sDiag);
IQ_stMeldung.sDiag	:= CONCAT(sConn,IQ_stMeldung.sDiag);

//****************************************************************************************************
// ENDE
END_ACTION

END_FUNCTION_BLOCK

// POUs/DiagSafety/FB_TwinSAFEConnInfo5Byte
(* Version history:
Description: Ethercat-Saftey Diagnose
Date          | Version    | created under        | Author          | Remark 
---------------------------------------------------------------------------------------- 
12/09/2011    | 1.1.0      | V2.11.0 (Build 1551)	| T.Löhner        | first release
25/04/2018    | 1.1.1      | V3.1.4022					| B.Daut				| bugfix und weitere Fehlermeldung hinzugefügt
02/12/2020    | 2.0.0      | V3.1.4024.10				| B.Daut				| für die EL1918 mit 8 Eingängen und 5 Byte ConnectionInfo
*)
FUNCTION_BLOCK FB_TwinSAFEConnInfo5Byte
VAR_OUTPUT
	Q_bErrorDiag	: BOOL;
	Q_bErrorState	: BOOL;
	Q_sDiag			: Tc2_System.T_MaxString;
	Q_sState			: Tc2_System.T_MaxString;
	Q_sState2		: Tc2_System.T_MaxString;
END_VAR

VAR_INPUT
	I_stInfoData			: ST_TwinSAFEConnInfo5Byte;
	I_nGrpId					: INT	:= 1;
	I_bGroupDeaktivated	: BOOL;	// Wenn die TwinSAFE-Gruppe deaktiviert wurde, darf die Connection kein Meldung absetzen
	I_nConnId				: INT;
	I_sConnName				: Tc2_System.T_MaxString;
END_VAR

VAR
	sConn				: Tc2_System.T_MaxString;;
	nDiag				: WORD;
	sStateOld		: Tc2_System.T_MaxString;
	sDiagOld			: Tc2_System.T_MaxString;
	tonStateChange	: TON;
	tonDiagChange	: TON;
END_VAR

//****************************************************************************************************
a_Info();

//****************************************************************************************************
// ENDE

ACTION a_Info:
// TwinSAFE-Connection
//****************************************************************************************************
Q_bErrorState		:= FALSE;
Q_bErrorDiag		:= FALSE;
Q_sState				:= '';
Q_sState2			:= '';
Q_sDiag				:= '';

sConn	:= CONCAT('Gruppe',INT_TO_STRING(I_nGrpId));
sConn	:= CONCAT(sConn,' => ');
sConn	:= CONCAT(sConn,'Connection');
sConn	:= CONCAT(sConn,INT_TO_STRING(I_nConnId));
sConn	:= CONCAT(sConn,' ');
sConn	:= CONCAT(sConn,I_sConnName);
sConn	:= CONCAT(sConn,' => ');

//****************************************************************************************************
// Klartext aus der Doku zur EL6900 PDF, Seite 16 oben, Tabelle 2-5

// State
CASE I_stInfoData.nMapState
OF

100: 	Q_sState 			:='Reset';
		Q_sState2			:='Der Zustand Reset dient dazu, nach dem Power-On oder einem Safety over EtherCAT Kommunikationsfehler die Safety over EtherCAT Connection neu zu initialisieren.';

101: 	Q_sState 			:='Session';
		Q_sState2			:='Beim Übergang in den bzw. im Zustand Session wird eine Session ID vom Safety over EtherCAT Master zum Safety over EtherCAT Slave übertragen, der wiederum mit einer eigenen Session ID antwortet.';

102: 	Q_sState 			:='Connection';
		Q_sState2			:='Im Zustand Connection wird eine Connection ID vom Safety over EtherCAT Master zum Safety over EtherCAT Slave übertragen.';

103: 	Q_sState 			:='Parameter';
		Q_sState2			:='Im Zustand Parameter werden sichere Kommunikations- und gerätespezifische Anwendungsparameter übertragen.';

104: 	Q_sState 			:='Data';
		Q_sState2			:='Im Zustand Data werden solange Safety over EtherCAT Cycles übertragen, bis entweder ein Kommunikationsfehler auftritt oder ein Safety over EtherCAT Node lokal gestoppt wird.';

105: 	Q_sState 			:='Shutdown';
		Q_sState2			:='Im Zustand Shutdown ist die Verbindung durch einen der Kommunikationspartner heruntergefahren worden.';

106: 	Q_sState 			:='Shutdown-Deactive';
		Q_sState2			:='Connection wurde über deactivate inputs heruntergefahren.';

ELSE
	Q_sState 			:='undefiniert';
	Q_sState2			:='';
	b_State();
END_CASE

//****************************************************************************************************
// Klartext aus der Doku zur EL6900 PDF, Seite 15 unten, Tabelle 2-4

// Diagnose

// Die Fehlerbits 0-3 kommen parallel, können also als Zahlen abgefragt werden
CASE I_stInfoData.nMapDiag OF
		0: ;
ELSE
	nDiag	:=UINT_TO_WORD(I_stInfoData.nMapDiag) AND 16#000F;
	CASE nDiag OF
		1: Q_sDiag			:='Ungueltiges Kommando';
			c_Diag();

		2: Q_sDiag 			:='Unbekanntes Kommando';
			c_Diag();

		3: Q_sDiag 			:='Ungueltige Connection ID';
			c_Diag();

		4: Q_sDiag 			:='Ungueltige CRC';
			c_Diag();

		5: Q_sDiag 			:='Watchdog abgelaufen';
			c_Diag();

		6: Q_sDiag 			:='Ungueltige FSoE address';
			c_Diag();

		7: Q_sDiag 			:='Ungueltige Daten';
			c_Diag();

		8: Q_sDiag 			:='Ungueltige Kommunikationsparameterlaenge';
			c_Diag();

		9: Q_sDiag 			:='Ungueltige Kommunikationsparameter';
			c_Diag();

		10:Q_sDiag 			:='Ungueltige Anwenderparameterlaenge';
			c_Diag();

		11:Q_sDiag 			:='Ungueltige Anwenderparameter';
			c_Diag();

		12:Q_sDiag		 	:='FSoE Master Reset';
			c_Diag();

		13:Q_sDiag		 	:='Modulfehler auf Slave erkannt, bei aktivierter "Option Modulfehler" ist ComError';
			c_Diag();

		14:Q_sDiag		 	:='Modulfehler auf EL29xx erkannt, bei aktivierter Option "Error acknowledge active"';
			c_Diag();

		15:Q_sDiag		 	:='Slave noch nicht gestartet, oder unerwartetes Fehlerargument';
			c_Diag();
	END_CASE

// Die Fehlerbits 4-7 kommen einzeln und müssen daher auch einzeln abgefragt werden.
	nDiag	:=UINT_TO_WORD(I_stInfoData.nMapDiag) AND 16#00F0;

	IF nDiag.4
	THEN
		Q_sDiag	:= 'Fehler beim FSoE Slave erkannt';
		c_Diag();
	ELSIF nDiag.5
	THEN
		Q_sDiag	:='FSoE Slave meldet Failsafe Value aktiv';
		c_Diag();
	ELSIF nDiag.6
	THEN
		Q_sDiag	:='StartUp';
		c_Diag();
	ELSIF nDiag.7
	THEN
		Q_sDiag	:='FSoE Master meldet Failsafe Value aktiv';
		c_Diag();
	END_IF

END_CASE

//****************************************************************************************************
// ENDE
END_ACTION

ACTION b_State:
//****************************************************************************************************
// Stateänderungen feststellen
IF Q_sState<> sStateOld
	OR I_bGroupDeaktivated
THEN
	Q_bErrorState	:= FALSE;
ELSE
	Q_bErrorState	:= TRUE;
END_IF

tonStateChange(
	IN	:= NOT Q_bErrorState,
	PT	:= T#500MS
);

IF tonStateChange.Q
THEN
	sStateOld	:= Q_sState;
END_IF

Q_sState	:= CONCAT('Status: ',Q_sState);
Q_sState	:= CONCAT(sConn,Q_sState);

//****************************************************************************************************
// ENDE
END_ACTION

ACTION c_Diag:
//****************************************************************************************************
// Diagänderungen feststellen
IF Q_sDiag<> sDiagOld
THEN
	Q_bErrorDiag	:= FALSE;
ELSE
	Q_bErrorDiag	:= TRUE;
END_IF

tonDiagChange(
	IN	:= NOT Q_bErrorDiag,
	PT	:= T#500MS
);

IF tonDiagChange.Q
THEN
	sDiagOld	:= Q_sDiag;
END_IF

Q_sDiag	:= CONCAT('Diagnose: ',Q_sDiag);
Q_sDiag	:= CONCAT(sConn,Q_sDiag);

//****************************************************************************************************
// ENDE
END_ACTION

END_FUNCTION_BLOCK

// POUs/DiagSafety/FB_TwinSAFEConnInfo5Byte_1
(* Version history:
Description: Ethercat-Saftey Diagnose
Date			| Version	| created under			| Author          | Remark 
---------------------------------------------------------------------------------------- 
12/09/2011	| 1.1.0		| V2.11.0 (Build 1551)	| T.Löhner        | first release
25/04/2018	| 1.1.1		| V3.1.4022					| B.Daut				| bugfix und weitere Fehlermeldung hinzugefügt
02/12/2020	| 2.0.0		| V3.1.4024.10				| B.Daut				| für die EL1918 mit 8 Eingängen und 5 Byte ConnectionInfo
28.02.2023	| 2.1.0		| V3.1.4024.40				| B.Daut				| Adaptiert für Avalon-HMI Meldesystem
*)
FUNCTION_BLOCK FB_TwinSAFEConnInfo5Byte_1
VAR_IN_OUT
	IQ_stMeldung			: ST_MeldSafetyOuts;
END_VAR
VAR_INPUT
	I_stInfoData			: ST_TwinSAFEConnInfo5Byte;
	I_nGrpId					: INT	:= 1;	// TwinSAFE-Gruppe zur Erstellung der Fehlermeldung
	I_bGroupDeaktivated	: BOOL;	// Wenn die TwinSAFE-Gruppe deaktiviert wurde, darf die Connection kein Meldung absetzen
	I_nConnId				: INT;	// TwinSAFE-ConnectionID zur Erstellung der Fehlermeldung
	I_sConnName				: Tc2_System.T_MaxString;	// TwinSAFE-ConnectionName zur Erstellung der Fehlermeldung
END_VAR
VAR
	sConn						: Tc2_System.T_MaxString;;
	nDiag						: WORD;
	sStateOld				: Tc2_System.T_MaxString;	// Zum feststellen einer Änderung und damit einhergehenden Neuauslösung der Meldung
	sDiagOld					: Tc2_System.T_MaxString;	// Zum feststellen einer Änderung und damit einhergehenden Neuauslösung der Meldung
	tonStateChange			: Tc2_Standard.TON;	// Zum feststellen einer Änderung und damit einhergehenden Neuauslösung der Meldung
	tonDiagChange			: Tc2_Standard.TON;	// Zum feststellen einer Änderung und damit einhergehenden Neuauslösung der Meldung
END_VAR

//****************************************************************************************************
a_Info();

//****************************************************************************************************
// ENDE

ACTION a_Info:
// TwinSAFE-Connection
//****************************************************************************************************
IQ_stMeldung.bMeldState		:= FALSE;
IQ_stMeldung.bMeldDiag		:= FALSE;
IQ_stMeldung.sState			:= '';
IQ_stMeldung.sDiag			:= '';

sConn	:= CONCAT('Gruppe',INT_TO_STRING(I_nGrpId));
sConn	:= CONCAT(sConn,' => ');
sConn	:= CONCAT(sConn,'Connection');
sConn	:= CONCAT(sConn,INT_TO_STRING(I_nConnId));
sConn	:= CONCAT(sConn,' ');
sConn	:= CONCAT(sConn,I_sConnName);
sConn	:= CONCAT(sConn,' => ');

//****************************************************************************************************
// Klartext aus der Doku zur EL6900 PDF, Seite 16 oben, Tabelle 2-5

// State
CASE I_stInfoData.nMapState
OF

100: 	IQ_stMeldung.sState	:='Reset: ';
		IQ_stMeldung.sState	:=CONCAT (IQ_stMeldung.sState,'Der Zustand Reset dient dazu, nach dem Power-On oder einem Safety over EtherCAT Kommunikationsfehler die Safety over EtherCAT Connection neu zu initialisieren.');

101: 	IQ_stMeldung.sState	:='Session: ';
		IQ_stMeldung.sState	:=CONCAT (IQ_stMeldung.sState,'Beim Übergang in den bzw. im Zustand Session wird eine Session ID vom Safety over EtherCAT Master zum Safety over EtherCAT Slave übertragen, der wiederum mit einer eigenen Session ID antwortet.');

102: 	IQ_stMeldung.sState	:='Connection: ';
		IQ_stMeldung.sState	:=CONCAT (IQ_stMeldung.sState,'Im Zustand Connection wird eine Connection ID vom Safety over EtherCAT Master zum Safety over EtherCAT Slave übertragen.');

103: 	IQ_stMeldung.sState	:='Parameter: ';
		IQ_stMeldung.sState	:=CONCAT (IQ_stMeldung.sState,'Im Zustand Parameter werden sichere Kommunikations- und gerätespezifische Anwendungsparameter übertragen.');

104: 	IQ_stMeldung.sState	:='Data: ';
		IQ_stMeldung.sState	:=CONCAT (IQ_stMeldung.sState,'Im Zustand Data werden solange Safety over EtherCAT Cycles übertragen, bis entweder ein Kommunikationsfehler auftritt oder ein Safety over EtherCAT Node lokal gestoppt wird.');

105: 	IQ_stMeldung.sState	:='Shutdown: ';
		IQ_stMeldung.sState	:=CONCAT (IQ_stMeldung.sState,'Im Zustand Shutdown ist die Verbindung durch einen der Kommunikationspartner heruntergefahren worden.');

106: 	IQ_stMeldung.sState	:='Shutdown-Deactive: ';
		IQ_stMeldung.sState	:=CONCAT (IQ_stMeldung.sState,'Connection wurde über deactivate inputs heruntergefahren.');

ELSE
	IQ_stMeldung.sState 			:='undefiniert';
	IQ_stMeldung.sState			:='';
	b_State();
END_CASE

//****************************************************************************************************
// Klartext aus der Doku zur EL6900 PDF, Seite 15 unten, Tabelle 2-4

// Diagnose

// Die Fehlerbits 0-3 kommen parallel, können also als Zahlen abgefragt werden
CASE I_stInfoData.nMapDiag OF
		0: ;
ELSE
	nDiag	:=UINT_TO_WORD(I_stInfoData.nMapDiag) AND 16#000F;
	CASE nDiag OF
		1: IQ_stMeldung.sDiag	:='Ungueltiges Kommando';
			c_Diag();

		2: IQ_stMeldung.sDiag	:='Unbekanntes Kommando';
			c_Diag();

		3: IQ_stMeldung.sDiag	:='Ungueltige Connection ID';
			c_Diag();

		4: IQ_stMeldung.sDiag	:='Ungueltige CRC';
			c_Diag();

		5: IQ_stMeldung.sDiag	:='Watchdog abgelaufen';
			c_Diag();

		6: IQ_stMeldung.sDiag	:='Ungueltige FSoE address';
			c_Diag();

		7: IQ_stMeldung.sDiag	:='Ungueltige Daten';
			c_Diag();

		8: IQ_stMeldung.sDiag	:='Ungueltige Kommunikationsparameterlaenge';
			c_Diag();

		9: IQ_stMeldung.sDiag	:='Ungueltige Kommunikationsparameter';
			c_Diag();

		10:IQ_stMeldung.sDiag	:='Ungueltige Anwenderparameterlaenge';
			c_Diag();

		11:IQ_stMeldung.sDiag	:='Ungueltige Anwenderparameter';
			c_Diag();

		12:IQ_stMeldung.sDiag	:='FSoE Master Reset';
			c_Diag();

		13:IQ_stMeldung.sDiag	:='Modulfehler auf Slave erkannt, bei aktivierter "Option Modulfehler" ist ComError';
			c_Diag();

		14:IQ_stMeldung.sDiag	:='Modulfehler auf EL29xx erkannt, bei aktivierter Option "Error acknowledge active"';
			c_Diag();

		15:IQ_stMeldung.sDiag	:='Slave noch nicht gestartet, oder unerwartetes Fehlerargument';
			c_Diag();
	END_CASE

// Die Fehlerbits 4-7 kommen einzeln und müssen daher auch einzeln abgefragt werden.
	nDiag	:=UINT_TO_WORD(I_stInfoData.nMapDiag) AND 16#00F0;

	IF nDiag.4
	THEN
		IQ_stMeldung.sDiag	:= 'Fehler beim FSoE Slave erkannt';
		c_Diag();
	ELSIF nDiag.5
	THEN
		IQ_stMeldung.sDiag	:='FSoE Slave meldet Failsafe Value aktiv';
		c_Diag();
	ELSIF nDiag.6
	THEN
		IQ_stMeldung.sDiag	:='StartUp';
		c_Diag();
	ELSIF nDiag.7
	THEN
		IQ_stMeldung.sDiag	:='FSoE Master meldet Failsafe Value aktiv';
		c_Diag();
	END_IF

END_CASE

//****************************************************************************************************
// ENDE
END_ACTION

ACTION b_State:
//****************************************************************************************************
// Stateänderungen feststellen
IF IQ_stMeldung.sState<> sStateOld
THEN
	IQ_stMeldung.bMeldState	:= FALSE;
ELSE
	IQ_stMeldung.bMeldState	:= NOT I_bGroupDeaktivated;
END_IF

tonStateChange(
	IN	:= NOT IQ_stMeldung.bMeldState,
	PT	:= T#500MS
);

IF tonStateChange.Q
THEN
	sStateOld	:= IQ_stMeldung.sState;
END_IF

IQ_stMeldung.sState	:= CONCAT('Status: ',IQ_stMeldung.sState);
IQ_stMeldung.sState	:= CONCAT(sConn,IQ_stMeldung.sState);

//****************************************************************************************************
// ENDE
END_ACTION

ACTION c_Diag:
//****************************************************************************************************
// Diagänderungen feststellen
IF IQ_stMeldung.sDiag<> sDiagOld
THEN
	IQ_stMeldung.bMeldDiag	:= FALSE;
ELSE
	IQ_stMeldung.bMeldDiag	:= NOT I_bGroupDeaktivated;
END_IF

tonDiagChange(
	IN	:= NOT IQ_stMeldung.bMeldDiag,
	PT	:= T#500MS
);

IF tonDiagChange.Q
THEN
	sDiagOld	:= IQ_stMeldung.sDiag;
END_IF

IQ_stMeldung.sDiag	:= CONCAT('Diagnose: ',IQ_stMeldung.sDiag);
IQ_stMeldung.sDiag	:= CONCAT(sConn,IQ_stMeldung.sDiag);

//****************************************************************************************************
// ENDE
END_ACTION

END_FUNCTION_BLOCK

// POUs/DiagSafety/FB_TwinSAFEConnInfoBasis
(* Version history:
Description: Ethercat-Saftey Diagnose
Date			| Version	| created under			| Author          | Remark 
---------------------------------------------------------------------------------------- 
12/09/2011	| 1.1.0		| V2.11.0 (Build 1551)	| T.Löhner        | first release
25/04/2018	| 1.1.1		| V2.11.0 (Build 4022)	| B.Daut				| bugfix und weitere Fehlermeldung hinzugefügt
28.02.2023	| 2.1.0		| V3.1.4024.40				| B.Daut				| Adaptiert für Avalon-HMI Meldesystem
05.01.2024	| 2.1.1		| V3.1.4024.54				| B.Daut				| Basisbaustein für alle Connections. Es ist ja nur das State und Diag notwendig.
*)
FUNCTION_BLOCK FB_TwinSAFEConnInfoBasis
VAR_IN_OUT
	IQ_stMeldung			: ST_MeldSafetyOuts;
END_VAR
VAR_INPUT
	I_stInfoData			: ST_TwinSAFE_ConnInfoBasis;
	I_nGrpId					: INT	:= 1;	// TwinSAFE-Gruppe zur Erstellung der Fehlermeldung
	I_bGroupDeaktivated	: BOOL;	// Wenn die TwinSAFE-Gruppe deaktiviert wurde, darf die Connection kein Meldung absetzen
	I_nConnId				: INT;	// TwinSAFE-ConnectionID zur Erstellung der Fehlermeldung
	I_sConnName				: Tc2_System.T_MaxString;	// TwinSAFE-ConnectionName zur Erstellung der Fehlermeldung
END_VAR
VAR
	sConn						: Tc2_System.T_MaxString;
	nDiag						: WORD;
	sStateOld				: Tc2_System.T_MaxString;	// Zum feststellen einer Änderung und damit einhergehenden Neuauslösung der Meldung
	sDiagOld					: Tc2_System.T_MaxString;	// Zum feststellen einer Änderung und damit einhergehenden Neuauslösung der Meldung
	tonStateChange			: Tc2_Standard.TON;	// Zum feststellen einer Änderung und damit einhergehenden Neuauslösung der Meldung
	tonDiagChange			: Tc2_Standard.TON;	// Zum feststellen einer Änderung und damit einhergehenden Neuauslösung der Meldung
END_VAR

//****************************************************************************************************
a_Info();

//****************************************************************************************************
// ENDE

ACTION a_Info:
// TwinSAFE-Connection
//****************************************************************************************************
IQ_stMeldung.bMeldState	:= FALSE;
IQ_stMeldung.bMeldDiag	:= FALSE;
IQ_stMeldung.sState		:= '';
IQ_stMeldung.sDiag		:= '';

sConn				:= CONCAT('Gruppe',INT_TO_STRING(I_nGrpId));
sConn				:= CONCAT(sConn,' => ');
sConn				:= CONCAT(sConn,'Connection');
sConn				:= CONCAT(sConn,INT_TO_STRING(I_nConnId));
sConn				:= CONCAT(sConn,' ');
sConn				:= CONCAT(sConn,I_sConnName);
sConn				:= CONCAT(sConn,' => ');

//****************************************************************************************************
// Klartext aus der Doku zur EL6900 PDF, Seite 16 oben, Tabelle 2-5

// State
CASE I_stInfoData.nMapState
OF

100: 	IQ_stMeldung.sState	:='Reset';
		IQ_stMeldung.sState	:=CONCAT (IQ_stMeldung.sState,'Der Zustand Reset dient dazu, nach dem Power-On oder einem Safety over EtherCAT Kommunikationsfehler die Safety over EtherCAT Connection neu zu initialisieren.');

101: 	IQ_stMeldung.sState	:='Session';
		IQ_stMeldung.sState	:=CONCAT (IQ_stMeldung.sState,'Beim Übergang in den bzw. im Zustand Session wird eine Session ID vom Safety over EtherCAT Master zum Safety over EtherCAT Slave übertragen, der wiederum mit einer eigenen Session ID antwortet.');

102: 	IQ_stMeldung.sState	:='Connection';
		IQ_stMeldung.sState	:=CONCAT (IQ_stMeldung.sState,'Im Zustand Connection wird eine Connection ID vom Safety over EtherCAT Master zum Safety over EtherCAT Slave übertragen.');

103: 	IQ_stMeldung.sState	:='Parameter';
		IQ_stMeldung.sState	:=CONCAT (IQ_stMeldung.sState,'Im Zustand Parameter werden sichere Kommunikations- und gerätespezifische Anwendungsparameter übertragen.');

104: 	IQ_stMeldung.sState	:='Data';
		IQ_stMeldung.sState	:=CONCAT (IQ_stMeldung.sState,'Im Zustand Data werden solange Safety over EtherCAT Cycles übertragen, bis entweder ein Kommunikationsfehler auftritt oder ein Safety over EtherCAT Node lokal gestoppt wird.');

105: 	IQ_stMeldung.sState	:='Shutdown';
		IQ_stMeldung.sState	:=CONCAT (IQ_stMeldung.sState,'Im Zustand Shutdown ist die Verbindung durch einen der Kommunikationspartner heruntergefahren worden.');

ELSE
	IQ_stMeldung.sState	:='undefiniert';
	//IQ_stMeldung.sState	:='';	// Warum war das hier drin??
	b_State();
END_CASE

//****************************************************************************************************
// Klartext aus der Doku zur EL6900 PDF, Seite 15 unten, Tabelle 2-4

// Diagnose

// Die Fehlerbits 0-3 kommen parallel, können also als Zahlen abgefragt werden
CASE I_stInfoData.nMapDiag OF
		0: ;
ELSE
	nDiag	:=UINT_TO_WORD(I_stInfoData.nMapDiag) AND 16#000F;
	CASE nDiag OF
		1: IQ_stMeldung.sDiag	:='Ungueltiges Kommando';
			c_Diag();

		2: IQ_stMeldung.sDiag	:='Unbekanntes Kommando';
			c_Diag();

		3: IQ_stMeldung.sDiag	:='Ungueltige Connection ID';
			c_Diag();

		4: IQ_stMeldung.sDiag	:='Ungueltige CRC';
			c_Diag();

		5: IQ_stMeldung.sDiag	:='Watchdog abgelaufen';
			c_Diag();

		6: IQ_stMeldung.sDiag	:='Ungueltige FSoE address';
			c_Diag();

		7: IQ_stMeldung.sDiag	:='Ungueltige data';
			c_Diag();

		8: IQ_stMeldung.sDiag	:='Ungueltige Kommunikationsparameterlaenge';
			c_Diag();

		9: IQ_stMeldung.sDiag	:='Ungueltige Kommunikationsparameter';
			c_Diag();

		10:IQ_stMeldung.sDiag	:='Ungueltige Anwenderparameterlaenge';
			c_Diag();

		11:IQ_stMeldung.sDiag	:='Ungueltige Anwenderparameter';
			c_Diag();

		12:IQ_stMeldung.sDiag	:='FSoE Master Reset';
			c_Diag();

		13:IQ_stMeldung.sDiag	:='Modulfehler auf Slave erkannt, bei aktivierter "Option Modulfehler" ist ComError';
			c_Diag();

		14:IQ_stMeldung.sDiag	:='Modulfehler auf EL290x erkannt, bei aktivierter Option "Error acknowledge active"';
			c_Diag();

		15:IQ_stMeldung.sDiag	:='Slave noch nicht gestartet, oder unerwartetes Fehlerargument';
			c_Diag();
	END_CASE

// Die Fehlerbits 4-7 kommen einzeln und müssen daher auch einzeln abgefragt werden.
	nDiag	:=UINT_TO_WORD(I_stInfoData.nMapDiag) AND 16#00F0;

	IF nDiag.4
	THEN
		IQ_stMeldung.sDiag	:= 'Fehler beim FSoE Slave erkannt';
		c_Diag();
	ELSIF nDiag.5
	THEN
		IQ_stMeldung.sDiag	:='FSoE Slave meldet Failsafe Value aktiv';
		c_Diag();
	ELSIF nDiag.6
	THEN
		IQ_stMeldung.sDiag	:='StartUp';
		c_Diag();
	ELSIF nDiag.7
	THEN
		IQ_stMeldung.sDiag	:='FSoE Master meldet Failsafe Value aktiv';
		c_Diag();
	END_IF

END_CASE

//****************************************************************************************************
// ENDE
END_ACTION

ACTION b_State:
//****************************************************************************************************
// Stateänderungen feststellen
IF IQ_stMeldung.sState<> sStateOld
THEN
	IQ_stMeldung.bMeldState	:= FALSE;
ELSE
	IQ_stMeldung.bMeldState	:= NOT I_bGroupDeaktivated;
END_IF

tonStateChange(
	IN	:= NOT IQ_stMeldung.bMeldState,
	PT	:= T#500MS
);

IF tonStateChange.Q
THEN
	sStateOld	:= IQ_stMeldung.sState;
END_IF

IQ_stMeldung.sState	:= CONCAT('Status: ',IQ_stMeldung.sState);
IQ_stMeldung.sState	:= CONCAT(sConn,IQ_stMeldung.sState);

//****************************************************************************************************
// ENDE
END_ACTION

ACTION c_Diag:
//****************************************************************************************************
// Diagänderungen feststellen
IF IQ_stMeldung.sDiag<> sDiagOld
THEN
	IQ_stMeldung.bMeldDiag	:= FALSE;
ELSE
	IQ_stMeldung.bMeldDiag	:= NOT I_bGroupDeaktivated;
END_IF

tonDiagChange(
	IN	:= NOT IQ_stMeldung.bMeldDiag,
	PT	:= T#500MS
);

IF tonDiagChange.Q
THEN
	sDiagOld	:= IQ_stMeldung.sDiag;
END_IF

IQ_stMeldung.sDiag	:= CONCAT('Diagnose: ',IQ_stMeldung.sDiag);
IQ_stMeldung.sDiag	:= CONCAT(sConn,IQ_stMeldung.sDiag);

//****************************************************************************************************
// ENDE
END_ACTION

END_FUNCTION_BLOCK

// POUs/DiagSafety/FB_TwinSAFEFBsInfo
(* Version History:
Description: Ethercat-Saftey Diagnose für TwinSAFE-FBs
Date			| Version	| created under			| Author				| Remark 
---------------------------------------------------------------------------------------- 
12/09/2011	| 1.1.0		| V2.11.0 (Build 1551)	| T.Löhner			| first release
28.02.2023	| 1.2.0		| V3.1.4024.40				| B.Daut				| Adaptiert für Avalon-HMI Meldesystem
*)
FUNCTION_BLOCK FB_TwinSAFEFBsInfo
VAR_IN_OUT
	IQ_stMeldung				: ST_MeldSafetyFBErrors;
END_VAR
VAR_INPUT
	I_stInfoData				: ST_TwinSAFE_FB_Info;	// TwinSAFE-Verbindung zu den TwinSAFE-FB
	I_nGrpId						: INT;	// TwinSAFE-Gruppe zur Erstellung der Fehlermeldung
	I_nFBId						: INT;	// TwinSAFE-FB-ID zur Erstellung der Fehlermeldung
	I_sFBName					: STRING;	// Name des Funktionsbausteins zur Erstellung der Fehlermeldung
	
	I_bMeldungFreigaben	: BOOL;	// TwinSAFE-FB darf überwacht werden. z.B. bFehlerEtherCATAllg
	
	I_sNameEinGruppe1			: STRING;	// Bezeichung der beiden Safety-Inputs der 1.FB-Eingangsgruppe 		=> bei EStop/MachineMonitoring/ConnectionShutdown/Muting/TwoHand
	I_sNameEinGruppe2			: STRING;	// Bezeichung der beiden Safety-Inputs der 2.FB-Eingangsgruppe 		=> bei EStop/MachineMonitoring/ConnectionShutdown/Muting/TwoHand
	I_sNameEinGruppe3			: STRING;	// Bezeichung der beiden Safety-Inputs der 3.FB-Eingangsgruppe 		=> bei EStop/MachineMonitoring/ConnectionShutdown/Muting/TwoHand
	I_sNameEinGruppe4			: STRING;	// Bezeichung der beiden Safety-Inputs der 4.FB-Eingangsgruppe 		=> bei EStop/MachineMonitoring/ConnectionShutdown/Muting/TwoHand
	I_sNameSecGruppe			: STRING;	// Bezeichung der beiden Safety-Inputs der FB-Secure-Eingangsgruppe 	=> bei MachineMonitoring
	I_sNameEMD1					: STRING;	// Bezeichung des Safety-Inputs für den Rückführkreis EDM1 				=> bei EStop/MachineMonitoring/Muting
	I_sNameEMD2					: STRING;	// Bezeichung des Safety-Inputs für den Rückführkreis EDM2 				=> bei EStop/MachineMonitoring/Muting
	I_sNameOSSDEinGruppe		: STRING;	// Bezeichung des Safety-Inputs für die OSSD-Eingangsgruppe				=> bei Muting
END_VAR
VAR
	sFB					: STRING;
	sState_old			: Tc2_System.T_MaxString;	// Zum feststellen einer Änderung und damit einhergehenden Neuauslösung der Meldung
	sDiag_old			: Tc2_System.T_MaxString;	// Zum feststellen einer Änderung und damit einhergehenden Neuauslösung der Meldung
	tonStateChange		: Tc2_Standard.TON;	// Zum feststellen einer Änderung und damit einhergehenden Neuauslösung der Meldung
	tonDiagChange		: Tc2_Standard.TON;	// Zum feststellen einer Änderung und damit einhergehenden Neuauslösung der Meldung
END_VAR

	(* ========================================================= *)
	;
	(* ========================================================= *)
	(* Aktionsaufrufe erfolgen je nach Art des TwinSAFE-Funktions-
		bausteins beim Aufruf von diesem FB *)

ACTION act_Diag:

	IF IQ_stMeldung.sMeldFBError_ErrorDiag<> sDiag_old THEN
		IQ_stMeldung.bMeldFBError_ErrorDiag	:= FALSE;
	ELSE
		IQ_stMeldung.bMeldFBError_ErrorDiag	:= I_bMeldungFreigaben;
	END_IF

	tonDiagChange(
		IN:= NOT IQ_stMeldung.bMeldFBError_ErrorDiag,
		PT:=t#500ms);

	IF tonDiagChange.Q THEN
		sDiag_old	:= IQ_stMeldung.sMeldFBError_ErrorDiag;
	END_IF

	IQ_stMeldung.sMeldFBError_ErrorDiag	:= CONCAT('Diagnose: ',IQ_stMeldung.sMeldFBError_ErrorDiag);
	IQ_stMeldung.sMeldFBError_ErrorDiag	:= CONCAT(sFB,IQ_stMeldung.sMeldFBError_ErrorDiag);

	(*BE*)
END_ACTION

ACTION act_State:

	IF IQ_stMeldung.sMeldFBError_ErrorState<> sState_old THEN
		IQ_stMeldung.bMeldFBError_ErrorState	:= FALSE;
	ELSE
		IQ_stMeldung.bMeldFBError_ErrorState	:= I_bMeldungFreigaben;
	END_IF

	tonStateChange(
		IN:= NOT IQ_stMeldung.bMeldFBError_ErrorState,
		PT:=t#500ms);

	IF tonStateChange.Q THEN
		sState_old	:= IQ_stMeldung.sMeldFBError_ErrorState;
	END_IF

	IQ_stMeldung.sMeldFBError_ErrorState	:= CONCAT('Status: ',IQ_stMeldung.sMeldFBError_ErrorState);
	IQ_stMeldung.sMeldFBError_ErrorState	:= CONCAT(sFB,IQ_stMeldung.sMeldFBError_ErrorState);

	(*BE*)
END_ACTION

ACTION actInfoAND:
	(* TwinSAFE-Funktionsbaustein FB AND*)
	(* ========================================================= *)

